LIN {X 0,Y 298.512,Z 418.3,A -85,B 0,C 180,E1 -16399.655,E2 -16399.655} C_VEL
LIN {X 0,Y 298.459,Z 418.309,A -85,B 0,C 180,E1 -16403.598,E2 -16403.598} C_VEL
LIN {X 0,Y 298.488,Z 418.301,A -85,B 0,C 180,E1 -16406.575,E2 -16406.575} C_VEL
LIN {X 0,Y 298.422,Z 418.314,A -85,B 0,C 180,E1 -16409.641,E2 -16409.641} C_VEL
LIN {X 0,Y 298.397,Z 418.313,A -85,B 0,C 180,E1 -16412.8,E2 -16412.8} C_VEL
LIN {X 0,Y 298.466,Z 418.305,A -85,B 0,C 180,E1 -16416.813,E2 -16416.813} C_VEL
LIN {X 0,Y 298.389,Z 418.316,A -85,B 0,C 180,E1 -16421.088,E2 -16421.088} C_VEL
LIN {X 0,Y 298.39,Z 418.318,A -85,B 0,C 180,E1 -16425.042,E2 -16425.042} C_VEL
LIN {X 0,Y 298.389,Z 418.318,A -85,B 0,C 180,E1 -16428.912,E2 -16428.912} C_VEL
LIN {X 0,Y 298.346,Z 418.518,A -85,B 0,C 180,E1 -16432.232,E2 -16432.232} C_VEL
LIN {X 0,Y 298.431,Z 421.494,A -85,B 0,C 180,E1 -16435.584,E2 -16435.584} C_VEL
LIN {X 0,Y 298.189,Z 424.493,A -85,B 0,C 180,E1 -16438.767,E2 -16438.767} C_VEL
LIN {X 0,Y 297.917,Z 427.501,A -85,B 0,C 180,E1 -16441.848,E2 -16441.848} C_VEL
LIN {X 0,Y 297.628,Z 431.178,A -85,B 0,C 180,E1 -16445.445,E2 -16445.445} C_VEL
LIN {X 0,Y 302.039,Z 446.255,A -85,B 0,C 180,E1 -16446.588,E2 -16446.588} C_VEL
LIN {X 0,Y 304.749,Z 458.03,A -85,B 0,C 180,E1 -16447.66,E2 -16447.66} C_VEL
LIN {X 0,Y 306.511,Z 468.932,A -85,B 0,C 180,E1 -16448.83,E2 -16448.83} C_VEL
LIN {X 0,Y 306.054,Z 475.088,A -85,B 0,C 180,E1 -16449.501,E2 -16449.501} C_VEL
LIN {X 0,Y 304.604,Z 485.483,A -85,B 0,C 180,E1 -16450.805,E2 -16450.805} C_VEL
LIN {X 0,Y 303.128,Z 495.965,A -85,B 0,C 180,E1 -16452.458,E2 -16452.458} C_VEL
LIN {X 0,Y 301.615,Z 504.454,A -85,B 0,C 180,E1 -16454.11,E2 -16454.11} C_VEL
LIN {X 0,Y 300.15,Z 512.702,A -85,B 0,C 180,E1 -16456.113,E2 -16456.113} C_VEL
LIN {X 0,Y 299.112,Z 518.344,A -85,B 0,C 180,E1 -16457.792,E2 -16457.792} C_VEL
LIN {X 0,Y 298.123,Z 523.842,A -85,B 0,C 180,E1 -16459.816,E2 -16459.816} C_VEL
LIN {X 0,Y 297.45,Z 528.155,A -85,B 0,C 180,E1 -16461.85,E2 -16461.85} C_VEL
LIN {X 0,Y 297.118,Z 530.806,A -85,B 0,C 180,E1 -16463.447,E2 -16463.447} C_VEL
LIN {X 0,Y 296.785,Z 533.683,A -85,B 0,C 180,E1 -16465.926,E2 -16465.926} C_VEL
LIN {X 0,Y 296.536,Z 535.288,A -85,B 0,C 180,E1 -16468.642,E2 -16468.642} C_VEL
LIN {X 0,Y 296.526,Z 535.518,A -85,B 0,C 180,E1 -16470,E2 -16470} C_VEL
LIN {X 0,Y 296.535,Z 535.326,A -85,B 0,C 180,E1 -16471.358,E2 -16471.358} C_VEL
LIN {X 0,Y 296.78,Z 533.772,A -85,B 0,C 180,E1 -16474.074,E2 -16474.074} C_VEL
LIN {X 0,Y 297.085,Z 531.047,A -85,B 0,C 180,E1 -16476.497,E2 -16476.497} C_VEL
LIN {X 0,Y 297.636,Z 527.076,A -85,B 0,C 180,E1 -16478.829,E2 -16478.829} C_VEL
LIN {X 0,Y 298.406,Z 522.443,A -85,B 0,C 180,E1 -16480.86,E2 -16480.86} C_VEL
LIN {X 0,Y 299.641,Z 515.457,A -85,B 0,C 180,E1 -16483.22,E2 -16483.22} C_VEL
LIN {X 0,Y 301,Z 507.884,A -85,B 0,C 180,E1 -16485.229,E2 -16485.229} C_VEL
LIN {X 0,Y 302.714,Z 498.347,A -85,B 0,C 180,E1 -16487.218,E2 -16487.218} C_VEL
LIN {X 0,Y 304.138,Z 488.507,A -85,B 0,C 180,E1 -16488.876,E2 -16488.876} C_VEL
LIN {X 0,Y 305.739,Z 477.425,A -85,B 0,C 180,E1 -16490.346,E2 -16490.346} C_VEL
LIN {X 0,Y 306.611,Z 469.946,A -85,B 0,C 180,E1 -16491.163,E2 -16491.163} C_VEL
LIN {X 0,Y 304.932,Z 458.822,A -85,B 0,C 180,E1 -16492.374,E2 -16492.374} C_VEL
LIN {X 0,Y 302.205,Z 446.768,A -85,B 0,C 180,E1 -16493.484,E2 -16493.484} C_VEL
LIN {X 0,Y 298.409,Z 433.993,A -85,B 0,C 180,E1 -16494.464,E2 -16494.464} C_VEL
LIN {X 0,Y 297.651,Z 431.164,A -85,B 0,C 180,E1 -16494.685,E2 -16494.685} C_VEL
LIN {X 0,Y 297.91,Z 427.623,A -85,B 0,C 180,E1 -16498.153,E2 -16498.153} C_VEL
LIN {X 0,Y 298.255,Z 423.912,A -85,B 0,C 180,E1 -16501.973,E2 -16501.973} C_VEL
LIN {X 0,Y 298.453,Z 421.544,A -85,B 0,C 180,E1 -16504.494,E2 -16504.494} C_VEL
LIN {X 0,Y 298.4,Z 418.632,A -85,B 0,C 180,E1 -16507.761,E2 -16507.761} C_VEL
LIN {X 0,Y 298.395,Z 418.314,A -85,B 0,C 180,E1 -16509.489,E2 -16509.489} C_VEL
LIN {X 0,Y 298.401,Z 418.314,A -85,B 0,C 180,E1 -16513.103,E2 -16513.103} C_VEL
LIN {X 0,Y 298.405,Z 418.316,A -85,B 0,C 180,E1 -16516.921,E2 -16516.921} C_VEL
LIN {X 0,Y 298.417,Z 418.312,A -85,B 0,C 180,E1 -16521.003,E2 -16521.003} C_VEL
LIN {X 0,Y 298.435,Z 418.309,A -85,B 0,C 180,E1 -16523.932,E2 -16523.932} C_VEL
LIN {X 0,Y 298.398,Z 418.314,A -85,B 0,C 180,E1 -16527.983,E2 -16527.983} C_VEL
LIN {X 0,Y 298.465,Z 418.306,A -85,B 0,C 180,E1 -16531.904,E2 -16531.904} C_VEL
LIN {X 0,Y 298.488,Z 418.302,A -85,B 0,C 180,E1 -16534.924,E2 -16534.924} C_VEL
LIN {X 0,Y 298.46,Z 418.305,A -85,B 0,C 180,E1 -16539.316,E2 -16539.316} C_VEL
LIN {X 0,Y 298.54,Z 418.299,A -85,B 0,C 180,E1 -16542.179,E2 -16542.179} C_VEL
LIN {X 0,Y 298.567,Z 418.29,A -85,B 0,C 180,E1 -16545.385,E2 -16545.385} C_VEL
LIN {X 0,Y 298.597,Z 418.288,A -85,B 0,C 180,E1 -16549.147,E2 -16549.147} C_VEL
LIN {X 0,Y 298.759,Z 418.267,A -85,B 0,C 180,E1 -16551.251,E2 -16551.251} C_VEL
LIN {X 0,Y 298.045,Z 418.361,A -85,B 0,C 180,E1 -16552.375,E2 -16552.375} C_VEL
LIN {X 0,Y 295.086,Z 418.728,A -85,B 0,C 180,E1 -16554.203,E2 -16554.203} C_VEL
LIN {X 0,Y 292.685,Z 419.028,A -85,B 0,C 180,E1 -16555.687,E2 -16555.687} C_VEL
LIN {X 0,Y 291.79,Z 419.135,A -85,B 0,C 180,E1 -16556.838,E2 -16556.838} C_VEL
LIN {X 0,Y 291.788,Z 419.136,A -85,B 0,C 180,E1 -16557.227,E2 -16557.227} C_VEL
LIN {X 0,Y 291.968,Z 419.118,A -85,B 0,C 180,E1 -16560,E2 -16560} C_VEL
LIN {X 0,Y 291.791,Z 419.135,A -85,B 0,C 180,E1 -16562.761,E2 -16562.761} C_VEL
LIN {X 0,Y 291.749,Z 419.142,A -85,B 0,C 180,E1 -16566.918,E2 -16566.918} C_VEL
LIN {X 0,Y 291.632,Z 419.159,A -85,B 0,C 180,E1 -16569.712,E2 -16569.712} C_VEL
LIN {X 0,Y 291.526,Z 419.171,A -85,B 0,C 180,E1 -16573.95,E2 -16573.95} C_VEL
LIN {X 0,Y 291.49,Z 419.174,A -85,B 0,C 180,E1 -16576.818,E2 -16576.818} C_VEL
LIN {X 0,Y 291.453,Z 419.179,A -85,B 0,C 180,E1 -16579.875,E2 -16579.875} C_VEL
LIN {X 0,Y 291.402,Z 419.184,A -85,B 0,C 180,E1 -16584.205,E2 -16584.205} C_VEL
LIN {X 0,Y 291.421,Z 419.186,A -85,B 0,C 180,E1 -16587.272,E2 -16587.272} C_VEL
LIN {X 0,Y 291.336,Z 419.193,A -85,B 0,C 180,E1 -16590.437,E2 -16590.437} C_VEL
LIN {X 0,Y 291.347,Z 419.191,A -85,B 0,C 180,E1 -16593.698,E2 -16593.698} C_VEL
LIN {X 0,Y 291.379,Z 419.191,A -85,B 0,C 180,E1 -16597.254,E2 -16597.254} C_VEL
LIN {X 0,Y 291.335,Z 419.2,A -85,B 0,C 180,E1 -16600.642,E2 -16600.642} C_VEL
LIN {X 0,Y 291.402,Z 419.214,A -85,B 0,C 180,E1 -16603.08,E2 -16603.08} C_VEL
LIN {X 0,Y 291.905,Z 422.504,A -85,B 0,C 180,E1 -16606.244,E2 -16606.244} C_VEL
LIN {X 0,Y 292.649,Z 426.936,A -85,B 0,C 180,E1 -16610.218,E2 -16610.218} C_VEL
LIN {X 0,Y 293,Z 430.406,A -85,B 0,C 180,E1 -16613.154,E2 -16613.154} C_VEL
LIN {X 0,Y 292.811,Z 433.555,A -85,B 0,C 180,E1 -16615.664,E2 -16615.664} C_VEL
LIN {X 0,Y 291.901,Z 439.373,A -85,B 0,C 180,E1 -16620.084,E2 -16620.084} C_VEL
LIN {X 0,Y 291.299,Z 443.573,A -85,B 0,C 180,E1 -16623.212,E2 -16623.212} C_VEL
LIN {X 0,Y 291.037,Z 445.704,A -85,B 0,C 180,E1 -16624.777,E2 -16624.777} C_VEL
LIN {X 0,Y 294.355,Z 459.225,A -85,B 0,C 180,E1 -16625.698,E2 -16625.698} C_VEL
LIN {X 0,Y 296.525,Z 470.949,A -85,B 0,C 180,E1 -16626.687,E2 -16626.687} C_VEL
LIN {X 0,Y 297.887,Z 482.255,A -85,B 0,C 180,E1 -16627.822,E2 -16627.822} C_VEL
LIN {X 0,Y 298.494,Z 491.884,A -85,B 0,C 180,E1 -16628.957,E2 -16628.957} C_VEL
LIN {X 0,Y 296.757,Z 503.417,A -85,B 0,C 180,E1 -16630.457,E2 -16630.457} C_VEL
LIN {X 0,Y 295.242,Z 512.708,A -85,B 0,C 180,E1 -16631.973,E2 -16631.973} C_VEL
LIN {X 0,Y 293.838,Z 521.184,A -85,B 0,C 180,E1 -16633.678,E2 -16633.678} C_VEL
LIN {X 0,Y 292.333,Z 529.457,A -85,B 0,C 180,E1 -16635.734,E2 -16635.734} C_VEL
LIN {X 0,Y 291.102,Z 536.125,A -85,B 0,C 180,E1 -16637.804,E2 -16637.804} C_VEL
LIN {X 0,Y 290.23,Z 542.233,A -85,B 0,C 180,E1 -16640.241,E2 -16640.241} C_VEL
LIN {X 0,Y 289.729,Z 546.204,A -85,B 0,C 180,E1 -16642.333,E2 -16642.333} C_VEL
LIN {X 0,Y 289.479,Z 549.227,A -85,B 0,C 180,E1 -16644.506,E2 -16644.506} C_VEL
LIN {X 0,Y 289.439,Z 551.537,A -85,B 0,C 180,E1 -16647.216,E2 -16647.216} C_VEL
LIN {X 0,Y 289.415,Z 552.145,A -85,B 0,C 180,E1 -16648.608,E2 -16648.608} C_VEL
LIN {X 0,Y 289.437,Z 552.359,A -85,B 0,C 180,E1 -16650,E2 -16650} C_VEL
LIN {X 0,Y 289.415,Z 552.138,A -85,B 0,C 180,E1 -16651.391,E2 -16651.391} C_VEL
LIN {X 0,Y 289.439,Z 551.526,A -85,B 0,C 180,E1 -16652.783,E2 -16652.783} C_VEL
LIN {X 0,Y 289.458,Z 549.252,A -85,B 0,C 180,E1 -16655.451,E2 -16655.451} C_VEL
LIN {X 0,Y 289.728,Z 546.171,A -85,B 0,C 180,E1 -16657.667,E2 -16657.667} C_VEL
LIN {X 0,Y 290.23,Z 542.186,A -85,B 0,C 180,E1 -16659.759,E2 -16659.759} C_VEL
LIN {X 0,Y 291.101,Z 536.059,A -85,B 0,C 180,E1 -16662.195,E2 -16662.195} C_VEL
LIN {X 0,Y 292.333,Z 529.376,A -85,B 0,C 180,E1 -16664.266,E2 -16664.266} C_VEL
LIN {X 0,Y 293.84,Z 521.086,A -85,B 0,C 180,E1 -16666.322,E2 -16666.322} C_VEL
LIN {X 0,Y 295.241,Z 512.583,A -85,B 0,C 180,E1 -16668.026,E2 -16668.026} C_VEL
LIN {X 0,Y 296.742,Z 503.258,A -85,B 0,C 180,E1 -16669.544,E2 -16669.544} C_VEL
LIN {X 0,Y 298.332,Z 493.123,A -85,B 0,C 180,E1 -16670.874,E2 -16670.874} C_VEL
LIN {X 0,Y 298.023,Z 483.792,A -85,B 0,C 180,E1 -16671.985,E2 -16671.985} C_VEL
LIN {X 0,Y 296.647,Z 472.092,A -85,B 0,C 180,E1 -16673.183,E2 -16673.183} C_VEL
LIN {X 0,Y 294.435,Z 459.785,A -85,B 0,C 180,E1 -16674.232,E2 -16674.232} C_VEL
LIN {X 0,Y 291.115,Z 446.415,A -85,B 0,C 180,E1 -16675.161,E2 -16675.161} C_VEL
LIN {X 0,Y 291.029,Z 445.687,A -85,B 0,C 180,E1 -16675.21,E2 -16675.21} C_VEL
LIN {X 0,Y 291.734,Z 440.822,A -85,B 0,C 180,E1 -16678.804,E2 -16678.804} C_VEL
LIN {X 0,Y 292.478,Z 435.563,A -85,B 0,C 180,E1 -16682.752,E2 -16682.752} C_VEL
LIN {X 0,Y 292.995,Z 432.197,A -85,B 0,C 180,E1 -16685.358,E2 -16685.358} C_VEL
LIN {X 0,Y 292.862,Z 428.244,A -85,B 0,C 180,E1 -16688.604,E2 -16688.604} C_VEL
LIN {X 0,Y 292.266,Z 424.569,A -85,B 0,C 180,E1 -16691.803,E2 -16691.803} C_VEL
LIN {X 0,Y 291.576,Z 420.462,A -85,B 0,C 180,E1 -16695.653,E2 -16695.653} C_VEL
LIN {X 0,Y 291.376,Z 419.19,A -85,B 0,C 180,E1 -16696.928,E2 -16696.928} C_VEL
LIN {X 0,Y 291.354,Z 419.196,A -85,B 0,C 180,E1 -16701.158,E2 -16701.158} C_VEL
LIN {X 0,Y 291.362,Z 419.196,A -85,B 0,C 180,E1 -16704.626,E2 -16704.626} C_VEL
LIN {X 0,Y 291.371,Z 419.19,A -85,B 0,C 180,E1 -16707.951,E2 -16707.951} C_VEL
LIN {X 0,Y 291.378,Z 419.19,A -85,B 0,C 180,E1 -16711.158,E2 -16711.158} C_VEL
LIN {X 0,Y 291.413,Z 419.185,A -85,B 0,C 180,E1 -16714.272,E2 -16714.272} C_VEL
LIN {X 0,Y 291.383,Z 419.188,A -85,B 0,C 180,E1 -16717.3,E2 -16717.3} C_VEL
LIN {X 0,Y 291.459,Z 419.18,A -85,B 0,C 180,E1 -16720.27,E2 -16720.27} C_VEL
LIN {X 0,Y 291.556,Z 419.17,A -85,B 0,C 180,E1 -16724.624,E2 -16724.624} C_VEL
LIN {X 0,Y 291.54,Z 419.169,A -85,B 0,C 180,E1 -16728.881,E2 -16728.881} C_VEL
LIN {X 0,Y 291.71,Z 419.147,A -85,B 0,C 180,E1 -16731.689,E2 -16731.689} C_VEL
LIN {X 0,Y 291.632,Z 419.158,A -85,B 0,C 180,E1 -16734.468,E2 -16734.468} C_VEL
LIN {X 0,Y 291.891,Z 419.126,A -85,B 0,C 180,E1 -16738.62,E2 -16738.62} C_VEL
LIN {X 0,Y 291.891,Z 419.124,A -85,B 0,C 180,E1 -16741.38,E2 -16741.38} C_VEL
LIN {X 0,Y 291.748,Z 419.141,A -85,B 0,C 180,E1 -16746.918,E2 -16746.918} C_VEL
LIN {X 0,Y 291.631,Z 419.158,A -85,B 0,C 180,E1 -16749.712,E2 -16749.712} C_VEL
LIN {X 0,Y 291.525,Z 419.173,A -85,B 0,C 180,E1 -16753.95,E2 -16753.95} C_VEL
LIN {X 0,Y 291.488,Z 419.174,A -85,B 0,C 180,E1 -16756.818,E2 -16756.818} C_VEL
LIN {X 0,Y 291.452,Z 419.18,A -85,B 0,C 180,E1 -16759.875,E2 -16759.875} C_VEL
LIN {X 0,Y 291.402,Z 419.186,A -85,B 0,C 180,E1 -16764.205,E2 -16764.205} C_VEL
LIN {X 0,Y 291.422,Z 419.183,A -85,B 0,C 180,E1 -16767.272,E2 -16767.272} C_VEL
LIN {X 0,Y 291.339,Z 419.192,A -85,B 0,C 180,E1 -16770.437,E2 -16770.437} C_VEL
LIN {X 0,Y 291.346,Z 419.195,A -85,B 0,C 180,E1 -16773.698,E2 -16773.698} C_VEL
LIN {X 0,Y 291.396,Z 419.188,A -85,B 0,C 180,E1 -16777.259,E2 -16777.259} C_VEL
LIN {X 0,Y 291.336,Z 419.193,A -85,B 0,C 180,E1 -16780.642,E2 -16780.642} C_VEL
LIN {X 0,Y 291.315,Z 419.197,A -85,B 0,C 180,E1 -16784.397,E2 -16784.397} C_VEL
LIN {X 0,Y 291.328,Z 419.196,A -85,B 0,C 180,E1 -16788.404,E2 -16788.404} C_VEL
LIN {X 0,Y 291.333,Z 419.198,A -85,B 0,C 180,E1 -16791.155,E2 -16791.155} C_VEL
LIN {X 0,Y 291.384,Z 420.19,A -85,B 0,C 180,E1 -16792.916,E2 -16792.916} C_VEL
LIN {X 0,Y 291.348,Z 423.185,A -85,B 0,C 180,E1 -16796.302,E2 -16796.302} C_VEL
LIN {X 0,Y 291.076,Z 426.197,A -85,B 0,C 180,E1 -16799.533,E2 -16799.533} C_VEL
LIN {X 0,Y 290.783,Z 429.984,A -85,B 0,C 180,E1 -16803.414,E2 -16803.414} C_VEL
LIN {X 0,Y 290.64,Z 431.426,A -85,B 0,C 180,E1 -16804.844,E2 -16804.844} C_VEL
LIN {X 0,Y 294.476,Z 444.129,A -85,B 0,C 180,E1 -16805.803,E2 -16805.803} C_VEL
LIN {X 0,Y 297.706,Z 457.33,A -85,B 0,C 180,E1 -16807.026,E2 -16807.026} C_VEL
LIN {X 0,Y 299.647,Z 469.149,A -85,B 0,C 180,E1 -16808.321,E2 -16808.321} C_VEL
LIN {X 0,Y 299.789,Z 472.293,A -85,B 0,C 180,E1 -16808.693,E2 -16808.693} C_VEL
LIN {X 0,Y 298.214,Z 483.339,A -85,B 0,C 180,E1 -16810.018,E2 -16810.018} C_VEL
LIN {X 0,Y 297,Z 492.352,A -85,B 0,C 180,E1 -16811.384,E2 -16811.384} C_VEL
LIN {X 0,Y 295.405,Z 501.444,A -85,B 0,C 180,E1 -16813.056,E2 -16813.056} C_VEL
LIN {X 0,Y 293.703,Z 510.354,A -85,B 0,C 180,E1 -16815.094,E2 -16815.094} C_VEL
LIN {X 0,Y 292.368,Z 517.522,A -85,B 0,C 180,E1 -16817.153,E2 -16817.153} C_VEL
LIN {X 0,Y 291.463,Z 522.355,A -85,B 0,C 180,E1 -16818.878,E2 -16818.878} C_VEL
LIN {X 0,Y 290.623,Z 527.05,A -85,B 0,C 180,E1 -16820.957,E2 -16820.957} C_VEL
LIN {X 0,Y 290.035,Z 531.259,A -85,B 0,C 180,E1 -16823.463,E2 -16823.463} C_VEL
LIN {X 0,Y 289.706,Z 533.888,A -85,B 0,C 180,E1 -16825.827,E2 -16825.827} C_VEL
LIN {X 0,Y 289.457,Z 535.492,A -85,B 0,C 180,E1 -16828.609,E2 -16828.609} C_VEL
LIN {X 0,Y 289.444,Z 535.722,A -85,B 0,C 180,E1 -16830,E2 -16830} C_VEL
LIN {X 0,Y 289.457,Z 535.53,A -85,B 0,C 180,E1 -16831.391,E2 -16831.391} C_VEL
LIN {X 0,Y 289.558,Z 534.943,A -85,B 0,C 180,E1 -16832.783,E2 -16832.783} C_VEL
LIN {X 0,Y 289.701,Z 533.975,A -85,B 0,C 180,E1 -16834.174,E2 -16834.174} C_VEL
LIN {X 0,Y 290.01,Z 531.455,A -85,B 0,C 180,E1 -16836.494,E2 -16836.494} C_VEL
LIN {X 0,Y 290.621,Z 527.279,A -85,B 0,C 180,E1 -16839.044,E2 -16839.044} C_VEL
LIN {X 0,Y 291.438,Z 522.646,A -85,B 0,C 180,E1 -16841.123,E2 -16841.123} C_VEL
LIN {X 0,Y 292.7,Z 515.661,A -85,B 0,C 180,E1 -16843.539,E2 -16843.539} C_VEL
LIN {X 0,Y 294.166,Z 508.085,A -85,B 0,C 180,E1 -16845.592,E2 -16845.592} C_VEL
LIN {X 0,Y 295.941,Z 498.548,A -85,B 0,C 180,E1 -16847.625,E2 -16847.625} C_VEL
LIN {X 0,Y 297.437,Z 488.707,A -85,B 0,C 180,E1 -16849.318,E2 -16849.318} C_VEL
LIN {X 0,Y 299.088,Z 477.624,A -85,B 0,C 180,E1 -16850.819,E2 -16850.819} C_VEL
LIN {X 0,Y 299.869,Z 471.72,A -85,B 0,C 180,E1 -16851.482,E2 -16851.482} C_VEL
LIN {X 0,Y 298.272,Z 460.146,A -85,B 0,C 180,E1 -16852.798,E2 -16852.798} C_VEL
LIN {X 0,Y 295.511,Z 447.816,A -85,B 0,C 180,E1 -16853.997,E2 -16853.997} C_VEL
LIN {X 0,Y 291.757,Z 435.282,A -85,B 0,C 180,E1 -16855.013,E2 -16855.013} C_VEL
LIN {X 0,Y 290.636,Z 431.427,A -85,B 0,C 180,E1 -16855.277,E2 -16855.277} C_VEL
LIN {X 0,Y 290.946,Z 427.824,A -85,B 0,C 180,E1 -16858.889,E2 -16858.889} C_VEL
LIN {X 0,Y 291.256,Z 424.534,A -85,B 0,C 180,E1 -16862.376,E2 -16862.376} C_VEL
LIN {X 0,Y 291.414,Z 421.811,A -85,B 0,C 180,E1 -16865.367,E2 -16865.367} C_VEL
LIN {X 0,Y 291.408,Z 420.148,A -85,B 0,C 180,E1 -16867.262,E2 -16867.262} C_VEL
LIN {X 0,Y 291.33,Z 419.196,A -85,B 0,C 180,E1 -16868.846,E2 -16868.846} C_VEL
LIN {X 0,Y 291.322,Z 419.196,A -85,B 0,C 180,E1 -16872.492,E2 -16872.492} C_VEL
LIN {X 0,Y 291.321,Z 419.196,A -85,B 0,C 180,E1 -16876.364,E2 -16876.364} C_VEL
LIN {X 0,Y 291.39,Z 419.19,A -85,B 0,C 180,E1 -16880.517,E2 -16880.517} C_VEL
LIN {X 0,Y 291.428,Z 419.184,A -85,B 0,C 180,E1 -16882.922,E2 -16882.922} C_VEL
LIN {X 0,Y 291.347,Z 419.195,A -85,B 0,C 180,E1 -16886.302,E2 -16886.302} C_VEL
LIN {X 0,Y 291.389,Z 419.189,A -85,B 0,C 180,E1 -16890.26,E2 -16890.26} C_VEL
LIN {X 0,Y 291.417,Z 419.184,A -85,B 0,C 180,E1 -16894.272,E2 -16894.272} C_VEL
LIN {X 0,Y 291.391,Z 419.185,A -85,B 0,C 180,E1 -16897.3,E2 -16897.3} C_VEL
LIN {X 0,Y 291.461,Z 419.181,A -85,B 0,C 180,E1 -16900.27,E2 -16900.27} C_VEL
LIN {X 0,Y 291.558,Z 419.166,A -85,B 0,C 180,E1 -16904.624,E2 -16904.624} C_VEL
LIN {X 0,Y 291.54,Z 419.167,A -85,B 0,C 180,E1 -16908.881,E2 -16908.881} C_VEL
LIN {X 0,Y 291.712,Z 419.147,A -85,B 0,C 180,E1 -16911.688,E2 -16911.688} C_VEL
LIN {X 0,Y 291.633,Z 419.157,A -85,B 0,C 180,E1 -16914.468,E2 -16914.468} C_VEL
LIN {X 0,Y 291.788,Z 419.136,A -85,B 0,C 180,E1 -16917.227,E2 -16917.227} C_VEL
LIN {X 0,Y 291.322,Z 419.198,A -85,B 0,C 180,E1 -16918.38,E2 -16918.38} C_VEL
LIN {X 0,Y 289.826,Z 419.385,A -85,B 0,C 180,E1 -16919.512,E2 -16919.512} C_VEL
LIN {X 0,Y 285.996,Z 419.862,A -85,B 0,C 180,E1 -16921.782,E2 -16921.782} C_VEL
LIN {X 0,Y 284.788,Z 420.008,A -85,B 0,C 180,E1 -16922.963,E2 -16922.963} C_VEL
LIN {X 0,Y 284.636,Z 420.025,A -85,B 0,C 180,E1 -16923.365,E2 -16923.365} C_VEL
LIN {X 0,Y 284.701,Z 420.02,A -85,B 0,C 180,E1 -16927.09,E2 -16927.09} C_VEL
LIN {X 0,Y 284.57,Z 420.037,A -85,B 0,C 180,E1 -16929.955,E2 -16929.955} C_VEL
LIN {X 0,Y 284.485,Z 420.047,A -85,B 0,C 180,E1 -16934.303,E2 -16934.303} C_VEL
LIN {X 0,Y 284.428,Z 420.056,A -85,B 0,C 180,E1 -16937.248,E2 -16937.248} C_VEL
LIN {X 0,Y 284.381,Z 420.059,A -85,B 0,C 180,E1 -16940.242,E2 -16940.242} C_VEL
LIN {X 0,Y 284.371,Z 420.061,A -85,B 0,C 180,E1 -16943.875,E2 -16943.875} C_VEL
LIN {X 0,Y 284.396,Z 420.061,A -85,B 0,C 180,E1 -16947.172,E2 -16947.172} C_VEL
LIN {X 0,Y 284.296,Z 420.069,A -85,B 0,C 180,E1 -16951.274,E2 -16951.274} C_VEL
LIN {X 0,Y 284.343,Z 420.066,A -85,B 0,C 180,E1 -16955.348,E2 -16955.348} C_VEL
LIN {X 0,Y 284.314,Z 420.068,A -85,B 0,C 180,E1 -16958.169,E2 -16958.169} C_VEL
LIN {X 0,Y 284.334,Z 420.082,A -85,B 0,C 180,E1 -16962.586,E2 -16962.586} C_VEL
LIN {X 0,Y 284.944,Z 423.867,A -85,B 0,C 180,E1 -16966.322,E2 -16966.322} C_VEL
LIN {X 0,Y 285.669,Z 428.1,A -85,B 0,C 180,E1 -16970.234,E2 -16970.234} C_VEL
LIN {X 0,Y 285.981,Z 431.266,A -85,B 0,C 180,E1 -16972.98,E2 -16972.98} C_VEL
LIN {X 0,Y 285.797,Z 434.403,A -85,B 0,C 180,E1 -16975.556,E2 -16975.556} C_VEL
LIN {X 0,Y 284.913,Z 439.712,A -85,B 0,C 180,E1 -16979.695,E2 -16979.695} C_VEL
LIN {X 0,Y 284.161,Z 444.764,A -85,B 0,C 180,E1 -16983.565,E2 -16983.565} C_VEL
LIN {X 0,Y 284.075,Z 445.488,A -85,B 0,C 180,E1 -16984.114,E2 -16984.114} C_VEL
LIN {X 0,Y 287.266,Z 458.185,A -85,B 0,C 180,E1 -16985.007,E2 -16985.007} C_VEL
LIN {X 0,Y 289.635,Z 470.588,A -85,B 0,C 180,E1 -16986.086,E2 -16986.086} C_VEL
LIN {X 0,Y 291.063,Z 482.048,A -85,B 0,C 180,E1 -16987.273,E2 -16987.273} C_VEL
LIN {X 0,Y 291.69,Z 493.113,A -85,B 0,C 180,E1 -16988.628,E2 -16988.628} C_VEL
LIN {X 0,Y 289.859,Z 504.345,A -85,B 0,C 180,E1 -16990.157,E2 -16990.157} C_VEL
LIN {X 0,Y 288.164,Z 514.307,A -85,B 0,C 180,E1 -16991.884,E2 -16991.884} C_VEL
LIN {X 0,Y 286.702,Z 522.472,A -85,B 0,C 180,E1 -16993.626,E2 -16993.626} C_VEL
LIN {X 0,Y 285.188,Z 530.49,A -85,B 0,C 180,E1 -16995.733,E2 -16995.733} C_VEL
LIN {X 0,Y 283.993,Z 536.919,A -85,B 0,C 180,E1 -16997.857,E2 -16997.857} C_VEL
LIN {X 0,Y 283.2,Z 542.029,A -85,B 0,C 180,E1 -16999.996,E2 -16999.996} C_VEL
LIN {X 0,Y 282.685,Z 546.001,A -85,B 0,C 180,E1 -17002.141,E2 -17002.141} C_VEL
LIN {X 0,Y 282.37,Z 549.27,A -85,B 0,C 180,E1 -17004.608,E2 -17004.608} C_VEL
LIN {X 0,Y 282.346,Z 551.333,A -85,B 0,C 180,E1 -17007.146,E2 -17007.146} C_VEL
LIN {X 0,Y 282.338,Z 551.942,A -85,B 0,C 180,E1 -17008.573,E2 -17008.573} C_VEL
LIN {X 0,Y 282.357,Z 552.156,A -85,B 0,C 180,E1 -17010,E2 -17010} C_VEL
LIN {X 0,Y 282.338,Z 551.935,A -85,B 0,C 180,E1 -17011.426,E2 -17011.426} C_VEL
LIN {X 0,Y 282.346,Z 551.322,A -85,B 0,C 180,E1 -17012.853,E2 -17012.853} C_VEL
LIN {X 0,Y 282.35,Z 549.293,A -85,B 0,C 180,E1 -17015.349,E2 -17015.349} C_VEL
LIN {X 0,Y 282.685,Z 545.966,A -85,B 0,C 180,E1 -17017.859,E2 -17017.859} C_VEL
LIN {X 0,Y 283.2,Z 541.979,A -85,B 0,C 180,E1 -17020.004,E2 -17020.004} C_VEL
LIN {X 0,Y 284.129,Z 535.853,A -85,B 0,C 180,E1 -17022.5,E2 -17022.5} C_VEL
LIN {X 0,Y 285.44,Z 529.17,A -85,B 0,C 180,E1 -17024.618,E2 -17024.618} C_VEL
LIN {X 0,Y 287.017,Z 520.879,A -85,B 0,C 180,E1 -17026.721,E2 -17026.721} C_VEL
LIN {X 0,Y 288.474,Z 512.376,A -85,B 0,C 180,E1 -17028.464,E2 -17028.464} C_VEL
LIN {X 0,Y 290.051,Z 503.05,A -85,B 0,C 180,E1 -17030.014,E2 -17030.014} C_VEL
LIN {X 0,Y 291.649,Z 492.913,A -85,B 0,C 180,E1 -17031.375,E2 -17031.375} C_VEL
LIN {X 0,Y 290.98,Z 481.79,A -85,B 0,C 180,E1 -17032.733,E2 -17032.733} C_VEL
LIN {X 0,Y 289.446,Z 469.456,A -85,B 0,C 180,E1 -17033.996,E2 -17033.996} C_VEL
LIN {X 0,Y 286.898,Z 456.681,A -85,B 0,C 180,E1 -17035.078,E2 -17035.078} C_VEL
LIN {X 0,Y 284.075,Z 445.463,A -85,B 0,C 180,E1 -17035.876,E2 -17035.876} C_VEL
LIN {X 0,Y 284.803,Z 440.618,A -85,B 0,C 180,E1 -17039.573,E2 -17039.573} C_VEL
LIN {X 0,Y 285.553,Z 435.93,A -85,B 0,C 180,E1 -17043.196,E2 -17043.196} C_VEL
LIN {X 0,Y 285.951,Z 432.253,A -85,B 0,C 180,E1 -17046.147,E2 -17046.147} C_VEL
LIN {X 0,Y 285.882,Z 429.93,A -85,B 0,C 180,E1 -17048.124,E2 -17048.124} C_VEL
LIN {X 0,Y 285.607,Z 427.452,A -85,B 0,C 180,E1 -17050.286,E2 -17050.286} C_VEL
LIN {X 0,Y 284.832,Z 423.147,A -85,B 0,C 180,E1 -17054.312,E2 -17054.312} C_VEL
LIN {X 0,Y 284.298,Z 420.073,A -85,B 0,C 180,E1 -17057.551,E2 -17057.551} C_VEL
LIN {X 0,Y 284.313,Z 420.072,A -85,B 0,C 180,E1 -17061.831,E2 -17061.831} C_VEL
LIN {X 0,Y 284.309,Z 420.072,A -85,B 0,C 180,E1 -17065.351,E2 -17065.351} C_VEL
LIN {X 0,Y 284.294,Z 420.075,A -85,B 0,C 180,E1 -17068.726,E2 -17068.726} C_VEL
LIN {X 0,Y 284.395,Z 420.062,A -85,B 0,C 180,E1 -17072.827,E2 -17072.827} C_VEL
LIN {X 0,Y 284.368,Z 420.065,A -85,B 0,C 180,E1 -17076.707,E2 -17076.707} C_VEL
LIN {X 0,Y 284.405,Z 420.057,A -85,B 0,C 180,E1 -17081.262,E2 -17081.262} C_VEL
LIN {X 0,Y 284.493,Z 420.049,A -85,B 0,C 180,E1 -17084.459,E2 -17084.459} C_VEL
LIN {X 0,Y 284.491,Z 420.049,A -85,B 0,C 180,E1 -17088.602,E2 -17088.602} C_VEL
LIN {X 0,Y 284.661,Z 420.024,A -85,B 0,C 180,E1 -17091.481,E2 -17091.481} C_VEL
LIN {X 0,Y 284.603,Z 420.033,A -85,B 0,C 180,E1 -17094.331,E2 -17094.331} C_VEL
LIN {X 0,Y 284.857,Z 420.002,A -85,B 0,C 180,E1 -17098.586,E2 -17098.586} C_VEL
LIN {X 0,Y 284.857,Z 420,A -85,B 0,C 180,E1 -17101.414,E2 -17101.414} C_VEL
LIN {X 0,Y 284.7,Z 420.019,A -85,B 0,C 180,E1 -17107.09,E2 -17107.09} C_VEL
LIN {X 0,Y 284.568,Z 420.04,A -85,B 0,C 180,E1 -17109.955,E2 -17109.955} C_VEL
LIN {X 0,Y 284.484,Z 420.048,A -85,B 0,C 180,E1 -17114.303,E2 -17114.303} C_VEL
LIN {X 0,Y 284.427,Z 420.054,A -85,B 0,C 180,E1 -17117.248,E2 -17117.248} C_VEL
LIN {X 0,Y 284.38,Z 420.06,A -85,B 0,C 180,E1 -17120.242,E2 -17120.242} C_VEL
LIN {X 0,Y 284.371,Z 420.064,A -85,B 0,C 180,E1 -17123.876,E2 -17123.876} C_VEL
LIN {X 0,Y 284.397,Z 420.058,A -85,B 0,C 180,E1 -17127.173,E2 -17127.173} C_VEL
LIN {X 0,Y 284.297,Z 420.071,A -85,B 0,C 180,E1 -17131.274,E2 -17131.274} C_VEL
LIN {X 0,Y 284.363,Z 420.064,A -85,B 0,C 180,E1 -17135.354,E2 -17135.354} C_VEL
LIN {X 0,Y 284.325,Z 420.067,A -85,B 0,C 180,E1 -17138.167,E2 -17138.167} C_VEL
LIN {X 0,Y 284.271,Z 420.074,A -85,B 0,C 180,E1 -17142.125,E2 -17142.125} C_VEL
LIN {X 0,Y 284.27,Z 420.075,A -85,B 0,C 180,E1 -17146.192,E2 -17146.192} C_VEL
LIN {X 0,Y 284.307,Z 420.071,A -85,B 0,C 180,E1 -17150.024,E2 -17150.024} C_VEL
LIN {X 0,Y 284.285,Z 420.385,A -85,B 0,C 180,E1 -17151.827,E2 -17151.827} C_VEL
LIN {X 0,Y 284.356,Z 423.38,A -85,B 0,C 180,E1 -17155.357,E2 -17155.357} C_VEL
LIN {X 0,Y 284.108,Z 426.398,A -85,B 0,C 180,E1 -17158.703,E2 -17158.703} C_VEL
LIN {X 0,Y 283.808,Z 429.451,A -85,B 0,C 180,E1 -17161.933,E2 -17161.933} C_VEL
LIN {X 0,Y 283.671,Z 431.624,A -85,B 0,C 180,E1 -17164.175,E2 -17164.175} C_VEL
LIN {X 0,Y 287.749,Z 445.057,A -85,B 0,C 180,E1 -17165.244,E2 -17165.244} C_VEL
LIN {X 0,Y 290.784,Z 457.397,A -85,B 0,C 180,E1 -17166.434,E2 -17166.434} C_VEL
LIN {X 0,Y 292.622,Z 467.644,A -85,B 0,C 180,E1 -17167.587,E2 -17167.587} C_VEL
LIN {X 0,Y 293.138,Z 472.504,A -85,B 0,C 180,E1 -17168.185,E2 -17168.185} C_VEL
LIN {X 0,Y 291.562,Z 483.547,A -85,B 0,C 180,E1 -17169.542,E2 -17169.542} C_VEL
LIN {X 0,Y 290.196,Z 493.082,A -85,B 0,C 180,E1 -17171.028,E2 -17171.028} C_VEL
LIN {X 0,Y 288.301,Z 503.272,A -85,B 0,C 180,E1 -17172.991,E2 -17172.991} C_VEL
LIN {X 0,Y 286.59,Z 511.889,A -85,B 0,C 180,E1 -17175.079,E2 -17175.079} C_VEL
LIN {X 0,Y 285.237,Z 518.756,A -85,B 0,C 180,E1 -17177.188,E2 -17177.188} C_VEL
LIN {X 0,Y 284.167,Z 524.253,A -85,B 0,C 180,E1 -17179.31,E2 -17179.31} C_VEL
LIN {X 0,Y 283.397,Z 528.565,A -85,B 0,C 180,E1 -17181.443,E2 -17181.443} C_VEL
LIN {X 0,Y 282.923,Z 531.752,A -85,B 0,C 180,E1 -17183.53,E2 -17183.53} C_VEL
LIN {X 0,Y 282.63,Z 534.092,A -85,B 0,C 180,E1 -17185.722,E2 -17185.722} C_VEL
LIN {X 0,Y 282.493,Z 535.084,A -85,B 0,C 180,E1 -17187.148,E2 -17187.148} C_VEL
LIN {X 0,Y 282.364,Z 535.925,A -85,B 0,C 180,E1 -17190,E2 -17190} C_VEL
LIN {X 0,Y 282.38,Z 535.733,A -85,B 0,C 180,E1 -17191.426,E2 -17191.426} C_VEL
LIN {X 0,Y 282.491,Z 535.146,A -85,B 0,C 180,E1 -17192.852,E2 -17192.852} C_VEL
LIN {X 0,Y 282.625,Z 534.178,A -85,B 0,C 180,E1 -17194.278,E2 -17194.278} C_VEL
LIN {X 0,Y 282.942,Z 531.848,A -85,B 0,C 180,E1 -17196.504,E2 -17196.504} C_VEL
LIN {X 0,Y 283.397,Z 528.762,A -85,B 0,C 180,E1 -17198.557,E2 -17198.557} C_VEL
LIN {X 0,Y 284.13,Z 524.51,A -85,B 0,C 180,E1 -17200.691,E2 -17200.691} C_VEL
LIN {X 0,Y 285.386,Z 518.07,A -85,B 0,C 180,E1 -17203.167,E2 -17203.167} C_VEL
LIN {X 0,Y 286.765,Z 510.99,A -85,B 0,C 180,E1 -17205.276,E2 -17205.276} C_VEL
LIN {X 0,Y 288.552,Z 502.165,A -85,B 0,C 180,E1 -17207.359,E2 -17207.359} C_VEL
LIN {X 0,Y 290.088,Z 492.988,A -85,B 0,C 180,E1 -17209.115,E2 -17209.115} C_VEL
LIN {X 0,Y 291.674,Z 483.081,A -85,B 0,C 180,E1 -17210.634,E2 -17210.634} C_VEL
LIN {X 0,Y 293.119,Z 473.494,A -85,B 0,C 180,E1 -17211.817,E2 -17211.817} C_VEL
LIN {X 0,Y 292.163,Z 464.863,A -85,B 0,C 180,E1 -17212.865,E2 -17212.865} C_VEL
LIN {X 0,Y 289.961,Z 453.507,A -85,B 0,C 180,E1 -17214.084,E2 -17214.084} C_VEL
LIN {X 0,Y 286.608,Z 441.206,A -85,B 0,C 180,E1 -17215.21,E2 -17215.21} C_VEL
LIN {X 0,Y 283.661,Z 431.608,A -85,B 0,C 180,E1 -17215.968,E2 -17215.968} C_VEL
LIN {X 0,Y 284.021,Z 427.719,A -85,B 0,C 180,E1 -17219.995,E2 -17219.995} C_VEL
LIN {X 0,Y 284.25,Z 425.011,A -85,B 0,C 180,E1 -17222.953,E2 -17222.953} C_VEL
LIN {X 0,Y 284.38,Z 422.009,A -85,B 0,C 180,E1 -17226.379,E2 -17226.379} C_VEL
LIN {X 0,Y 284.311,Z 420.497,A -85,B 0,C 180,E1 -17228.169,E2 -17228.169} C_VEL
LIN {X 0,Y 284.307,Z 420.069,A -85,B 0,C 180,E1 -17229.995,E2 -17229.995} C_VEL
LIN {X 0,Y 284.268,Z 420.073,A -85,B 0,C 180,E1 -17234.195,E2 -17234.195} C_VEL
LIN {X 0,Y 284.275,Z 420.074,A -85,B 0,C 180,E1 -17238.125,E2 -17238.125} C_VEL
LIN {X 0,Y 284.338,Z 420.066,A -85,B 0,C 180,E1 -17242.274,E2 -17242.274} C_VEL
LIN {X 0,Y 284.326,Z 420.067,A -85,B 0,C 180,E1 -17245.353,E2 -17245.353} C_VEL
LIN {X 0,Y 284.298,Z 420.072,A -85,B 0,C 180,E1 -17248.726,E2 -17248.726} C_VEL
LIN {X 0,Y 284.398,Z 420.058,A -85,B 0,C 180,E1 -17252.827,E2 -17252.827} C_VEL
LIN {X 0,Y 284.371,Z 420.062,A -85,B 0,C 180,E1 -17256.707,E2 -17256.707} C_VEL
LIN {X 0,Y 284.406,Z 420.056,A -85,B 0,C 180,E1 -17261.262,E2 -17261.262} C_VEL
LIN {X 0,Y 284.495,Z 420.046,A -85,B 0,C 180,E1 -17264.459,E2 -17264.459} C_VEL
LIN {X 0,Y 284.491,Z 420.046,A -85,B 0,C 180,E1 -17268.601,E2 -17268.601} C_VEL
LIN {X 0,Y 284.662,Z 420.024,A -85,B 0,C 180,E1 -17271.481,E2 -17271.481} C_VEL
LIN {X 0,Y 284.604,Z 420.033,A -85,B 0,C 180,E1 -17274.331,E2 -17274.331} C_VEL
LIN {X 0,Y 284.857,Z 420,A -85,B 0,C 180,E1 -17278.586,E2 -17278.586} C_VEL
LIN {X 0,Y 284.858,Z 420.002,A -85,B 0,C 180,E1 -17281.414,E2 -17281.414} C_VEL
LIN {X 0,Y 284.636,Z 420.025,A -85,B 0,C 180,E1 -17283.365,E2 -17283.365} C_VEL
LIN {X 0,Y 283.856,Z 420.125,A -85,B 0,C 180,E1 -17284.546,E2 -17284.546} C_VEL
LIN {X 0,Y 281.064,Z 420.473,A -85,B 0,C 180,E1 -17286.475,E2 -17286.475} C_VEL
LIN {X 0,Y 277.932,Z 420.863,A -85,B 0,C 180,E1 -17288.842,E2 -17288.842} C_VEL
LIN {X 0,Y 277.563,Z 420.908,A -85,B 0,C 180,E1 -17289.659,E2 -17289.659} C_VEL
LIN {X 0,Y 277.438,Z 420.924,A -85,B 0,C 180,E1 -17294.674,E2 -17294.674} C_VEL
LIN {X 0,Y 277.347,Z 420.939,A -85,B 0,C 180,E1 -17299.234,E2 -17299.234} C_VEL
LIN {X 0,Y 277.321,Z 420.938,A -85,B 0,C 180,E1 -17304.17,E2 -17304.17} C_VEL
LIN {X 0,Y 277.325,Z 420.94,A -85,B 0,C 180,E1 -17307.504,E2 -17307.504} C_VEL
LIN {X 0,Y 277.274,Z 420.946,A -85,B 0,C 180,E1 -17310.481,E2 -17310.481} C_VEL
LIN {X 0,Y 277.249,Z 420.947,A -85,B 0,C 180,E1 -17313.896,E2 -17313.896} C_VEL
LIN {X 0,Y 277.27,Z 420.947,A -85,B 0,C 180,E1 -17317.469,E2 -17317.469} C_VEL
LIN {X 0,Y 277.258,Z 421.046,A -85,B 0,C 180,E1 -17322.165,E2 -17322.165} C_VEL
LIN {X 0,Y 277.759,Z 423.905,A -85,B 0,C 180,E1 -17325.111,E2 -17325.111} C_VEL
LIN {X 0,Y 278.453,Z 428.153,A -85,B 0,C 180,E1 -17329.217,E2 -17329.217} C_VEL
LIN {X 0,Y 278.968,Z 432.126,A -85,B 0,C 180,E1 -17332.798,E2 -17332.798} C_VEL
LIN {X 0,Y 278.791,Z 435.264,A -85,B 0,C 180,E1 -17335.445,E2 -17335.445} C_VEL
LIN {X 0,Y 277.887,Z 440.454,A -85,B 0,C 180,E1 -17339.614,E2 -17339.614} C_VEL
LIN {X 0,Y 277.134,Z 445.282,A -85,B 0,C 180,E1 -17343.417,E2 -17343.417} C_VEL
LIN {X 0,Y 279.782,Z 455.675,A -85,B 0,C 180,E1 -17344.164,E2 -17344.164} C_VEL
LIN {X 0,Y 282.423,Z 468.047,A -85,B 0,C 180,E1 -17345.243,E2 -17345.243} C_VEL
LIN {X 0,Y 284.058,Z 480.175,A -85,B 0,C 180,E1 -17346.499,E2 -17346.499} C_VEL
LIN {X 0,Y 284.86,Z 491.573,A -85,B 0,C 180,E1 -17347.912,E2 -17347.912} C_VEL
LIN {X 0,Y 284.677,Z 495.642,A -85,B 0,C 180,E1 -17348.455,E2 -17348.455} C_VEL
LIN {X 0,Y 282.75,Z 506.287,A -85,B 0,C 180,E1 -17350.015,E2 -17350.015} C_VEL
LIN {X 0,Y 281.186,Z 515.254,A -85,B 0,C 180,E1 -17351.66,E2 -17351.66} C_VEL
LIN {X 0,Y 279.573,Z 523.758,A -85,B 0,C 180,E1 -17353.572,E2 -17353.572} C_VEL
LIN {X 0,Y 278.04,Z 531.444,A -85,B 0,C 180,E1 -17355.732,E2 -17355.732} C_VEL
LIN {X 0,Y 277.001,Z 536.714,A -85,B 0,C 180,E1 -17357.546,E2 -17357.546} C_VEL
LIN {X 0,Y 276.186,Z 541.825,A -85,B 0,C 180,E1 -17359.739,E2 -17359.739} C_VEL
LIN {X 0,Y 275.617,Z 545.796,A -85,B 0,C 180,E1 -17361.938,E2 -17361.938} C_VEL
LIN {X 0,Y 275.263,Z 549.311,A -85,B 0,C 180,E1 -17364.714,E2 -17364.714} C_VEL
LIN {X 0,Y 275.256,Z 551.13,A -85,B 0,C 180,E1 -17367.073,E2 -17367.073} C_VEL
LIN {X 0,Y 275.263,Z 551.739,A -85,B 0,C 180,E1 -17368.537,E2 -17368.537} C_VEL
LIN {X 0,Y 275.278,Z 551.953,A -85,B 0,C 180,E1 -17370,E2 -17370} C_VEL
LIN {X 0,Y 275.263,Z 551.731,A -85,B 0,C 180,E1 -17371.463,E2 -17371.463} C_VEL
LIN {X 0,Y 275.255,Z 551.118,A -85,B 0,C 180,E1 -17372.927,E2 -17372.927} C_VEL
LIN {X 0,Y 275.253,Z 549.313,A -85,B 0,C 180,E1 -17375.262,E2 -17375.262} C_VEL
LIN {X 0,Y 275.616,Z 545.76,A -85,B 0,C 180,E1 -17378.062,E2 -17378.062} C_VEL
LIN {X 0,Y 276.186,Z 541.774,A -85,B 0,C 180,E1 -17380.261,E2 -17380.261} C_VEL
LIN {X 0,Y 277.171,Z 535.646,A -85,B 0,C 180,E1 -17382.819,E2 -17382.819} C_VEL
LIN {X 0,Y 278.563,Z 528.964,A -85,B 0,C 180,E1 -17384.987,E2 -17384.987} C_VEL
LIN {X 0,Y 280.208,Z 520.672,A -85,B 0,C 180,E1 -17387.14,E2 -17387.14} C_VEL
LIN {X 0,Y 281.697,Z 512.167,A -85,B 0,C 180,E1 -17388.925,E2 -17388.925} C_VEL
LIN {X 0,Y 283.57,Z 501.665,A -85,B 0,C 180,E1 -17390.681,E2 -17390.681} C_VEL
LIN {X 0,Y 284.842,Z 494.131,A -85,B 0,C 180,E1 -17391.722,E2 -17391.722} C_VEL
LIN {X 0,Y 284.33,Z 483.363,A -85,B 0,C 180,E1 -17393.103,E2 -17393.103} C_VEL
LIN {X 0,Y 282.906,Z 471.207,A -85,B 0,C 180,E1 -17394.418,E2 -17394.418} C_VEL
LIN {X 0,Y 280.355,Z 458.105,A -85,B 0,C 180,E1 -17395.613,E2 -17395.613} C_VEL
LIN {X 0,Y 277.127,Z 445.238,A -85,B 0,C 180,E1 -17396.588,E2 -17396.588} C_VEL
LIN {X 0,Y 277.991,Z 439.975,A -85,B 0,C 180,E1 -17400.732,E2 -17400.732} C_VEL
LIN {X 0,Y 278.792,Z 435.197,A -85,B 0,C 180,E1 -17404.555,E2 -17404.555} C_VEL
LIN {X 0,Y 278.915,Z 432.062,A -85,B 0,C 180,E1 -17407.21,E2 -17407.21} C_VEL
LIN {X 0,Y 278.48,Z 428.095,A -85,B 0,C 180,E1 -17410.79,E2 -17410.79} C_VEL
LIN {X 0,Y 277.691,Z 423.592,A -85,B 0,C 180,E1 -17415.125,E2 -17415.125} C_VEL
LIN {X 0,Y 277.236,Z 420.952,A -85,B 0,C 180,E1 -17418.024,E2 -17418.024} C_VEL
LIN {X 0,Y 277.269,Z 420.951,A -85,B 0,C 180,E1 -17422.531,E2 -17422.531} C_VEL
LIN {X 0,Y 277.248,Z 420.951,A -85,B 0,C 180,E1 -17426.104,E2 -17426.104} C_VEL
LIN {X 0,Y 277.262,Z 420.948,A -85,B 0,C 180,E1 -17429.539,E2 -17429.539} C_VEL
LIN {X 0,Y 277.357,Z 420.938,A -85,B 0,C 180,E1 -17432.864,E2 -17432.864} C_VEL
LIN {X 0,Y 277.329,Z 420.939,A -85,B 0,C 180,E1 -17436.08,E2 -17436.08} C_VEL
LIN {X 0,Y 277.346,Z 420.94,A -85,B 0,C 180,E1 -17440.766,E2 -17440.766} C_VEL
LIN {X 0,Y 277.436,Z 420.925,A -85,B 0,C 180,E1 -17445.326,E2 -17445.326} C_VEL
LIN {X 0,Y 277.509,Z 420.916,A -85,B 0,C 180,E1 -17449.789,E2 -17449.789} C_VEL
LIN {X 0,Y 277.655,Z 420.897,A -85,B 0,C 180,E1 -17452.729,E2 -17452.729} C_VEL
LIN {X 0,Y 277.823,Z 420.879,A -85,B 0,C 180,E1 -17458.551,E2 -17458.551} C_VEL
LIN {X 0,Y 277.823,Z 420.876,A -85,B 0,C 180,E1 -17461.45,E2 -17461.45} C_VEL
LIN {X 0,Y 277.655,Z 420.897,A -85,B 0,C 180,E1 -17467.271,E2 -17467.271} C_VEL
LIN {X 0,Y 277.509,Z 420.918,A -85,B 0,C 180,E1 -17470.211,E2 -17470.211} C_VEL
LIN {X 0,Y 277.437,Z 420.925,A -85,B 0,C 180,E1 -17474.674,E2 -17474.674} C_VEL
LIN {X 0,Y 277.346,Z 420.934,A -85,B 0,C 180,E1 -17479.234,E2 -17479.234} C_VEL
LIN {X 0,Y 277.321,Z 420.94,A -85,B 0,C 180,E1 -17484.171,E2 -17484.171} C_VEL
LIN {X 0,Y 277.326,Z 420.941,A -85,B 0,C 180,E1 -17487.505,E2 -17487.505} C_VEL
LIN {X 0,Y 277.273,Z 420.944,A -85,B 0,C 180,E1 -17490.481,E2 -17490.481} C_VEL
LIN {X 0,Y 277.256,Z 420.949,A -85,B 0,C 180,E1 -17493.895,E2 -17493.895} C_VEL
LIN {X 0,Y 277.283,Z 420.947,A -85,B 0,C 180,E1 -17497.467,E2 -17497.467} C_VEL
LIN {X 0,Y 277.211,Z 420.956,A -85,B 0,C 180,E1 -17501.237,E2 -17501.237} C_VEL
LIN {X 0,Y 277.218,Z 420.956,A -85,B 0,C 180,E1 -17505.223,E2 -17505.223} C_VEL
LIN {X 0,Y 277.224,Z 420.954,A -85,B 0,C 180,E1 -17509.512,E2 -17509.512} C_VEL
LIN {X 0,Y 277.227,Z 420.954,A -85,B 0,C 180,E1 -17510.671,E2 -17510.671} C_VEL
LIN {X 0,Y 277.32,Z 422.07,A -85,B 0,C 180,E1 -17512.539,E2 -17512.539} C_VEL
LIN {X 0,Y 277.349,Z 423.567,A -85,B 0,C 180,E1 -17514.351,E2 -17514.351} C_VEL
LIN {X 0,Y 277.147,Z 426.589,A -85,B 0,C 180,E1 -17517.824,E2 -17517.824} C_VEL
LIN {X 0,Y 276.834,Z 429.658,A -85,B 0,C 180,E1 -17521.161,E2 -17521.161} C_VEL
LIN {X 0,Y 276.697,Z 431.833,A -85,B 0,C 180,E1 -17523.459,E2 -17523.459} C_VEL
LIN {X 0,Y 281.142,Z 446.408,A -85,B 0,C 180,E1 -17524.695,E2 -17524.695} C_VEL
LIN {X 0,Y 284.22,Z 458.995,A -85,B 0,C 180,E1 -17525.975,E2 -17525.975} C_VEL
LIN {X 0,Y 286.034,Z 469.583,A -85,B 0,C 180,E1 -17527.233,E2 -17527.233} C_VEL
LIN {X 0,Y 286.395,Z 474.279,A -85,B 0,C 180,E1 -17527.834,E2 -17527.834} C_VEL
LIN {X 0,Y 284.718,Z 484.939,A -85,B 0,C 180,E1 -17529.217,E2 -17529.217} C_VEL
LIN {X 0,Y 283.163,Z 495.208,A -85,B 0,C 180,E1 -17530.91,E2 -17530.91} C_VEL
LIN {X 0,Y 281.537,Z 503.478,A -85,B 0,C 180,E1 -17532.569,E2 -17532.569} C_VEL
LIN {X 0,Y 279.745,Z 512.095,A -85,B 0,C 180,E1 -17534.705,E2 -17534.705} C_VEL
LIN {X 0,Y 278.322,Z 518.962,A -85,B 0,C 180,E1 -17536.864,E2 -17536.864} C_VEL
LIN {X 0,Y 277.18,Z 524.458,A -85,B 0,C 180,E1 -17539.038,E2 -17539.038} C_VEL
LIN {X 0,Y 276.387,Z 528.77,A -85,B 0,C 180,E1 -17541.224,E2 -17541.224} C_VEL
LIN {X 0,Y 275.832,Z 532.199,A -85,B 0,C 180,E1 -17543.564,E2 -17543.564} C_VEL
LIN {X 0,Y 275.557,Z 534.297,A -85,B 0,C 180,E1 -17545.612,E2 -17545.612} C_VEL
LIN {X 0,Y 275.427,Z 535.288,A -85,B 0,C 180,E1 -17547.075,E2 -17547.075} C_VEL
LIN {X 0,Y 275.286,Z 536.129,A -85,B 0,C 180,E1 -17550,E2 -17550} C_VEL
LIN {X 0,Y 275.306,Z 535.936,A -85,B 0,C 180,E1 -17551.463,E2 -17551.463} C_VEL
LIN {X 0,Y 275.425,Z 535.349,A -85,B 0,C 180,E1 -17552.925,E2 -17552.925} C_VEL
LIN {X 0,Y 275.552,Z 534.382,A -85,B 0,C 180,E1 -17554.388,E2 -17554.388} C_VEL
LIN {X 0,Y 275.872,Z 532.245,A -85,B 0,C 180,E1 -17556.51,E2 -17556.51} C_VEL
LIN {X 0,Y 276.386,Z 528.965,A -85,B 0,C 180,E1 -17558.776,E2 -17558.776} C_VEL
LIN {X 0,Y 277.148,Z 524.713,A -85,B 0,C 180,E1 -17560.964,E2 -17560.964} C_VEL
LIN {X 0,Y 278.483,Z 518.272,A -85,B 0,C 180,E1 -17563.5,E2 -17563.5} C_VEL
LIN {X 0,Y 279.917,Z 511.192,A -85,B 0,C 180,E1 -17565.659,E2 -17565.659} C_VEL
LIN {X 0,Y 281.796,Z 502.366,A -85,B 0,C 180,E1 -17567.789,E2 -17567.789} C_VEL
LIN {X 0,Y 283.433,Z 492.836,A -85,B 0,C 180,E1 -17569.649,E2 -17569.649} C_VEL
LIN {X 0,Y 285.231,Z 481.993,A -85,B 0,C 180,E1 -17571.312,E2 -17571.312} C_VEL
LIN {X 0,Y 286.451,Z 473.696,A -85,B 0,C 180,E1 -17572.352,E2 -17572.352} C_VEL
LIN {X 0,Y 284.81,Z 461.921,A -85,B 0,C 180,E1 -17573.808,E2 -17573.808} C_VEL
LIN {X 0,Y 282.226,Z 450.355,A -85,B 0,C 180,E1 -17575.046,E2 -17575.046} C_VEL
LIN {X 0,Y 278.546,Z 437.681,A -85,B 0,C 180,E1 -17576.198,E2 -17576.198} C_VEL
LIN {X 0,Y 276.715,Z 431.839,A -85,B 0,C 180,E1 -17576.659,E2 -17576.659} C_VEL
LIN {X 0,Y 277,Z 428.233,A -85,B 0,C 180,E1 -17580.493,E2 -17580.493} C_VEL
LIN {X 0,Y 277.282,Z 425.224,A -85,B 0,C 180,E1 -17583.891,E2 -17583.891} C_VEL
LIN {X 0,Y 277.341,Z 422.2,A -85,B 0,C 180,E1 -17587.458,E2 -17587.458} C_VEL
LIN {X 0,Y 277.235,Z 420.951,A -85,B 0,C 180,E1 -17589.328,E2 -17589.328} C_VEL
LIN {X 0,Y 277.219,Z 420.952,A -85,B 0,C 180,E1 -17593.197,E2 -17593.197} C_VEL
LIN {X 0,Y 277.22,Z 420.952,A -85,B 0,C 180,E1 -17597.324,E2 -17597.324} C_VEL
LIN {X 0,Y 277.278,Z 420.944,A -85,B 0,C 180,E1 -17601.79,E2 -17601.79} C_VEL
LIN {X 0,Y 277.306,Z 420.943,A -85,B 0,C 180,E1 -17604.344,E2 -17604.344} C_VEL
LIN {X 0,Y 277.247,Z 420.948,A -85,B 0,C 180,E1 -17607.837,E2 -17607.837} C_VEL
LIN {X 0,Y 277.273,Z 420.944,A -85,B 0,C 180,E1 -17611.21,E2 -17611.21} C_VEL
LIN {X 0,Y 277.315,Z 420.94,A -85,B 0,C 180,E1 -17614.48,E2 -17614.48} C_VEL
LIN {X 0,Y 277.293,Z 420.942,A -85,B 0,C 180,E1 -17617.655,E2 -17617.655} C_VEL
LIN {X 0,Y 277.348,Z 420.936,A -85,B 0,C 180,E1 -17620.766,E2 -17620.766} C_VEL
LIN {X 0,Y 277.437,Z 420.923,A -85,B 0,C 180,E1 -17625.326,E2 -17625.326} C_VEL
LIN {X 0,Y 277.509,Z 420.918,A -85,B 0,C 180,E1 -17629.789,E2 -17629.789} C_VEL
LIN {X 0,Y 277.656,Z 420.897,A -85,B 0,C 180,E1 -17632.729,E2 -17632.729} C_VEL
LIN {X 0,Y 277.823,Z 420.876,A -85,B 0,C 180,E1 -17638.55,E2 -17638.55} C_VEL
LIN {X 0,Y 277.824,Z 420.878,A -85,B 0,C 180,E1 -17641.449,E2 -17641.449} C_VEL
LIN {X 0,Y 277.656,Z 420.899,A -85,B 0,C 180,E1 -17647.271,E2 -17647.271} C_VEL
LIN {X 0,Y 277.563,Z 420.908,A -85,B 0,C 180,E1 -17649.659,E2 -17649.659} C_VEL
LIN {X 0,Y 276.804,Z 421.004,A -85,B 0,C 180,E1 -17650.868,E2 -17650.868} C_VEL
LIN {X 0,Y 273.923,Z 421.366,A -85,B 0,C 180,E1 -17652.839,E2 -17652.839} C_VEL
LIN {X 0,Y 271.519,Z 421.666,A -85,B 0,C 180,E1 -17654.44,E2 -17654.44} C_VEL
LIN {X 0,Y 270.47,Z 421.795,A -85,B 0,C 180,E1 -17655.68,E2 -17655.68} C_VEL
LIN {X 0,Y 270.372,Z 421.805,A -85,B 0,C 180,E1 -17656.101,E2 -17656.101} C_VEL
LIN {X 0,Y 270.295,Z 421.814,A -85,B 0,C 180,E1 -17660.602,E2 -17660.602} C_VEL
LIN {X 0,Y 270.276,Z 421.816,A -85,B 0,C 180,E1 -17664.585,E2 -17664.585} C_VEL
LIN {X 0,Y 270.271,Z 421.816,A -85,B 0,C 180,E1 -17667.909,E2 -17667.909} C_VEL
LIN {X 0,Y 270.186,Z 421.826,A -85,B 0,C 180,E1 -17671.348,E2 -17671.348} C_VEL
LIN {X 0,Y 270.204,Z 421.827,A -85,B 0,C 180,E1 -17674.905,E2 -17674.905} C_VEL
LIN {X 0,Y 270.199,Z 421.83,A -85,B 0,C 180,E1 -17678.71,E2 -17678.71} C_VEL
LIN {X 0,Y 270.223,Z 421.998,A -85,B 0,C 180,E1 -17681.717,E2 -17681.717} C_VEL
LIN {X 0,Y 270.825,Z 425.583,A -85,B 0,C 180,E1 -17685.52,E2 -17685.52} C_VEL
LIN {X 0,Y 271.524,Z 429.815,A -85,B 0,C 180,E1 -17689.677,E2 -17689.677} C_VEL
LIN {X 0,Y 271.931,Z 433.702,A -85,B 0,C 180,E1 -17693.244,E2 -17693.244} C_VEL
LIN {X 0,Y 271.619,Z 436.794,A -85,B 0,C 180,E1 -17695.892,E2 -17695.892} C_VEL
LIN {X 0,Y 270.657,Z 442.301,A -85,B 0,C 180,E1 -17700.438,E2 -17700.438} C_VEL
LIN {X 0,Y 270.176,Z 445.061,A -85,B 0,C 180,E1 -17702.673,E2 -17702.673} C_VEL
LIN {X 0,Y 273.654,Z 458.531,A -85,B 0,C 180,E1 -17703.721,E2 -17703.721} C_VEL
LIN {X 0,Y 276.118,Z 471.062,A -85,B 0,C 180,E1 -17704.914,E2 -17704.914} C_VEL
LIN {X 0,Y 277.559,Z 483.196,A -85,B 0,C 180,E1 -17706.274,E2 -17706.274} C_VEL
LIN {X 0,Y 278.118,Z 492.859,A -85,B 0,C 180,E1 -17707.551,E2 -17707.551} C_VEL
LIN {X 0,Y 277.619,Z 498.03,A -85,B 0,C 180,E1 -17708.27,E2 -17708.27} C_VEL
LIN {X 0,Y 275.681,Z 508.197,A -85,B 0,C 180,E1 -17709.869,E2 -17709.869} C_VEL
LIN {X 0,Y 274.04,Z 517,A -85,B 0,C 180,E1 -17711.604,E2 -17711.604} C_VEL
LIN {X 0,Y 272.443,Z 524.931,A -85,B 0,C 180,E1 -17713.515,E2 -17713.515} C_VEL
LIN {X 0,Y 270.916,Z 532.363,A -85,B 0,C 180,E1 -17715.733,E2 -17715.733} C_VEL
LIN {X 0,Y 269.708,Z 538.334,A -85,B 0,C 180,E1 -17717.968,E2 -17717.968} C_VEL
LIN {X 0,Y 268.947,Z 543.056,A -85,B 0,C 180,E1 -17720.22,E2 -17720.22} C_VEL
LIN {X 0,Y 268.421,Z 546.666,A -85,B 0,C 180,E1 -17722.477,E2 -17722.477} C_VEL
LIN {X 0,Y 268.179,Z 549.304,A -85,B 0,C 180,E1 -17724.775,E2 -17724.775} C_VEL
LIN {X 0,Y 268.168,Z 550.926,A -85,B 0,C 180,E1 -17726.995,E2 -17726.995} C_VEL
LIN {X 0,Y 268.189,Z 551.535,A -85,B 0,C 180,E1 -17728.498,E2 -17728.498} C_VEL
LIN {X 0,Y 268.202,Z 551.749,A -85,B 0,C 180,E1 -17730,E2 -17730} C_VEL
LIN {X 0,Y 268.189,Z 551.527,A -85,B 0,C 180,E1 -17731.501,E2 -17731.501} C_VEL
LIN {X 0,Y 268.167,Z 550.913,A -85,B 0,C 180,E1 -17733.004,E2 -17733.004} C_VEL
LIN {X 0,Y 268.169,Z 549.304,A -85,B 0,C 180,E1 -17735.2,E2 -17735.2} C_VEL
LIN {X 0,Y 268.562,Z 545.554,A -85,B 0,C 180,E1 -17738.275,E2 -17738.275} C_VEL
LIN {X 0,Y 269.17,Z 541.568,A -85,B 0,C 180,E1 -17740.531,E2 -17740.531} C_VEL
LIN {X 0,Y 270.228,Z 535.44,A -85,B 0,C 180,E1 -17743.154,E2 -17743.154} C_VEL
LIN {X 0,Y 271.701,Z 528.757,A -85,B 0,C 180,E1 -17745.375,E2 -17745.375} C_VEL
LIN {X 0,Y 273.415,Z 520.466,A -85,B 0,C 180,E1 -17747.579,E2 -17747.579} C_VEL
LIN {X 0,Y 274.958,Z 511.959,A -85,B 0,C 180,E1 -17749.407,E2 -17749.407} C_VEL
LIN {X 0,Y 276.948,Z 501.458,A -85,B 0,C 180,E1 -17751.199,E2 -17751.199} C_VEL
LIN {X 0,Y 278.097,Z 493.917,A -85,B 0,C 180,E1 -17752.276,E2 -17752.276} C_VEL
LIN {X 0,Y 277.515,Z 483.144,A -85,B 0,C 180,E1 -17753.704,E2 -17753.704} C_VEL
LIN {X 0,Y 276.069,Z 470.983,A -85,B 0,C 180,E1 -17755.064,E2 -17755.064} C_VEL
LIN {X 0,Y 273.535,Z 458.023,A -85,B 0,C 180,E1 -17756.29,E2 -17756.29} C_VEL
LIN {X 0,Y 270.201,Z 445.018,A -85,B 0,C 180,E1 -17757.327,E2 -17757.327} C_VEL
LIN {X 0,Y 271.022,Z 440.208,A -85,B 0,C 180,E1 -17761.24,E2 -17761.24} C_VEL
LIN {X 0,Y 271.771,Z 436.034,A -85,B 0,C 180,E1 -17764.675,E2 -17764.675} C_VEL
LIN {X 0,Y 271.901,Z 433.647,A -85,B 0,C 180,E1 -17766.748,E2 -17766.748} C_VEL
LIN {X 0,Y 271.746,Z 431.04,A -85,B 0,C 180,E1 -17769.116,E2 -17769.116} C_VEL
LIN {X 0,Y 271.174,Z 427.645,A -85,B 0,C 180,E1 -17772.364,E2 -17772.364} C_VEL
LIN {X 0,Y 270.461,Z 423.417,A -85,B 0,C 180,E1 -17776.684,E2 -17776.684} C_VEL
LIN {X 0,Y 270.184,Z 421.832,A -85,B 0,C 180,E1 -17778.483,E2 -17778.483} C_VEL
LIN {X 0,Y 270.207,Z 421.831,A -85,B 0,C 180,E1 -17781.374,E2 -17781.374} C_VEL
LIN {X 0,Y 270.203,Z 421.832,A -85,B 0,C 180,E1 -17785.095,E2 -17785.095} C_VEL
LIN {X 0,Y 270.201,Z 421.829,A -85,B 0,C 180,E1 -17789.131,E2 -17789.131} C_VEL
LIN {X 0,Y 270.264,Z 421.819,A -85,B 0,C 180,E1 -17792.146,E2 -17792.146} C_VEL
LIN {X 0,Y 270.278,Z 421.817,A -85,B 0,C 180,E1 -17795.519,E2 -17795.519} C_VEL
LIN {X 0,Y 270.303,Z 421.816,A -85,B 0,C 180,E1 -17800.245,E2 -17800.245} C_VEL
LIN {X 0,Y 270.405,Z 421.802,A -85,B 0,C 180,E1 -17804.935,E2 -17804.935} C_VEL
LIN {X 0,Y 270.444,Z 421.796,A -85,B 0,C 180,E1 -17809.519,E2 -17809.519} C_VEL
LIN {X 0,Y 270.613,Z 421.776,A -85,B 0,C 180,E1 -17812.539,E2 -17812.539} C_VEL
LIN {X 0,Y 270.789,Z 421.755,A -85,B 0,C 180,E1 -17818.513,E2 -17818.513} C_VEL
LIN {X 0,Y 270.789,Z 421.753,A -85,B 0,C 180,E1 -17821.487,E2 -17821.487} C_VEL
LIN {X 0,Y 270.613,Z 421.775,A -85,B 0,C 180,E1 -17827.461,E2 -17827.461} C_VEL
LIN {X 0,Y 270.444,Z 421.796,A -85,B 0,C 180,E1 -17830.481,E2 -17830.481} C_VEL
LIN {X 0,Y 270.405,Z 421.8,A -85,B 0,C 180,E1 -17835.065,E2 -17835.065} C_VEL
LIN {X 0,Y 270.303,Z 421.813,A -85,B 0,C 180,E1 -17839.756,E2 -17839.756} C_VEL
LIN {X 0,Y 270.275,Z 421.816,A -85,B 0,C 180,E1 -17844.586,E2 -17844.586} C_VEL
LIN {X 0,Y 270.271,Z 421.819,A -85,B 0,C 180,E1 -17847.909,E2 -17847.909} C_VEL
LIN {X 0,Y 270.186,Z 421.829,A -85,B 0,C 180,E1 -17851.348,E2 -17851.348} C_VEL
LIN {X 0,Y 270.216,Z 421.824,A -85,B 0,C 180,E1 -17854.904,E2 -17854.904} C_VEL
LIN {X 0,Y 270.223,Z 421.824,A -85,B 0,C 180,E1 -17858.717,E2 -17858.717} C_VEL
LIN {X 0,Y 270.173,Z 421.832,A -85,B 0,C 180,E1 -17863.251,E2 -17863.251} C_VEL
LIN {X 0,Y 270.176,Z 421.833,A -85,B 0,C 180,E1 -17867.443,E2 -17867.443} C_VEL
LIN {X 0,Y 270.175,Z 421.832,A -85,B 0,C 180,E1 -17869.434,E2 -17869.434} C_VEL
LIN {X 0,Y 270.246,Z 422.283,A -85,B 0,C 180,E1 -17871.381,E2 -17871.381} C_VEL
LIN {X 0,Y 270.277,Z 425.288,A -85,B 0,C 180,E1 -17875.106,E2 -17875.106} C_VEL
LIN {X 0,Y 270.011,Z 428.828,A -85,B 0,C 180,E1 -17879.199,E2 -17879.199} C_VEL
LIN {X 0,Y 269.689,Z 432.042,A -85,B 0,C 180,E1 -17882.716,E2 -17882.716} C_VEL
LIN {X 0,Y 274.137,Z 446.272,A -85,B 0,C 180,E1 -17883.976,E2 -17883.976} C_VEL
LIN {X 0,Y 276.928,Z 457.342,A -85,B 0,C 180,E1 -17885.132,E2 -17885.132} C_VEL
LIN {X 0,Y 279.052,Z 468.802,A -85,B 0,C 180,E1 -17886.514,E2 -17886.514} C_VEL
LIN {X 0,Y 279.734,Z 474.585,A -85,B 0,C 180,E1 -17887.289,E2 -17887.289} C_VEL
LIN {X 0,Y 277.902,Z 486.316,A -85,B 0,C 180,E1 -17888.877,E2 -17888.877} C_VEL
LIN {X 0,Y 276.18,Z 496.794,A -85,B 0,C 180,E1 -17890.682,E2 -17890.682} C_VEL
LIN {X 0,Y 274.418,Z 505.28,A -85,B 0,C 180,E1 -17892.487,E2 -17892.487} C_VEL
LIN {X 0,Y 272.623,Z 513.528,A -85,B 0,C 180,E1 -17894.679,E2 -17894.679} C_VEL
LIN {X 0,Y 271.423,Z 519.167,A -85,B 0,C 180,E1 -17896.524,E2 -17896.524} C_VEL
LIN {X 0,Y 270.207,Z 524.664,A -85,B 0,C 180,E1 -17898.751,E2 -17898.751} C_VEL
LIN {X 0,Y 269.35,Z 528.976,A -85,B 0,C 180,E1 -17900.993,E2 -17900.993} C_VEL
LIN {X 0,Y 268.751,Z 532.622,A -85,B 0,C 180,E1 -17903.58,E2 -17903.58} C_VEL
LIN {X 0,Y 268.486,Z 534.501,A -85,B 0,C 180,E1 -17905.496,E2 -17905.496} C_VEL
LIN {X 0,Y 268.362,Z 535.491,A -85,B 0,C 180,E1 -17906.998,E2 -17906.998} C_VEL
LIN {X 0,Y 268.21,Z 536.332,A -85,B 0,C 180,E1 -17910,E2 -17910} C_VEL
LIN {X 0,Y 268.234,Z 536.139,A -85,B 0,C 180,E1 -17911.502,E2 -17911.502} C_VEL
LIN {X 0,Y 268.36,Z 535.552,A -85,B 0,C 180,E1 -17913.003,E2 -17913.003} C_VEL
LIN {X 0,Y 268.481,Z 534.585,A -85,B 0,C 180,E1 -17914.504,E2 -17914.504} C_VEL
LIN {X 0,Y 268.791,Z 532.667,A -85,B 0,C 180,E1 -17916.495,E2 -17916.495} C_VEL
LIN {X 0,Y 269.348,Z 529.168,A -85,B 0,C 180,E1 -17919.007,E2 -17919.007} C_VEL
LIN {X 0,Y 270.18,Z 524.916,A -85,B 0,C 180,E1 -17921.25,E2 -17921.25} C_VEL
LIN {X 0,Y 271.59,Z 518.474,A -85,B 0,C 180,E1 -17923.849,E2 -17923.849} C_VEL
LIN {X 0,Y 273.094,Z 511.393,A -85,B 0,C 180,E1 -17926.06,E2 -17926.06} C_VEL
LIN {X 0,Y 275.057,Z 502.567,A -85,B 0,C 180,E1 -17928.24,E2 -17928.24} C_VEL
LIN {X 0,Y 276.689,Z 493.363,A -85,B 0,C 180,E1 -17930.085,E2 -17930.085} C_VEL
LIN {X 0,Y 278.437,Z 483.48,A -85,B 0,C 180,E1 -17931.663,E2 -17931.663} C_VEL
LIN {X 0,Y 279.75,Z 475.377,A -85,B 0,C 180,E1 -17932.722,E2 -17932.722} C_VEL
LIN {X 0,Y 278.426,Z 464.662,A -85,B 0,C 180,E1 -17934.131,E2 -17934.131} C_VEL
LIN {X 0,Y 275.879,Z 452.665,A -85,B 0,C 180,E1 -17935.498,E2 -17935.498} C_VEL
LIN {X 0,Y 272.348,Z 440.202,A -85,B 0,C 180,E1 -17936.712,E2 -17936.712} C_VEL
LIN {X 0,Y 269.704,Z 432.043,A -85,B 0,C 180,E1 -17937.411,E2 -17937.411} C_VEL
LIN {X 0,Y 270.023,Z 428.44,A -85,B 0,C 180,E1 -17941.369,E2 -17941.369} C_VEL
LIN {X 0,Y 270.298,Z 425.428,A -85,B 0,C 180,E1 -17944.892,E2 -17944.892} C_VEL
LIN {X 0,Y 270.255,Z 422.31,A -85,B 0,C 180,E1 -17948.725,E2 -17948.725} C_VEL
LIN {X 0,Y 270.171,Z 421.83,A -85,B 0,C 180,E1 -17951.028,E2 -17951.028} C_VEL
LIN {X 0,Y 270.168,Z 421.83,A -85,B 0,C 180,E1 -17955.383,E2 -17955.383} C_VEL
LIN {X 0,Y 270.177,Z 421.829,A -85,B 0,C 180,E1 -17959.434,E2 -17959.434} C_VEL
LIN {X 0,Y 270.257,Z 421.819,A -85,B 0,C 180,E1 -17963.722,E2 -17963.722} C_VEL
LIN {X 0,Y 270.207,Z 421.826,A -85,B 0,C 180,E1 -17966.893,E2 -17966.893} C_VEL
LIN {X 0,Y 270.199,Z 421.827,A -85,B 0,C 180,E1 -17970.383,E2 -17970.383} C_VEL
LIN {X 0,Y 270.265,Z 421.818,A -85,B 0,C 180,E1 -17973.764,E2 -17973.764} C_VEL
LIN {X 0,Y 270.239,Z 421.821,A -85,B 0,C 180,E1 -17977.039,E2 -17977.039} C_VEL
LIN {X 0,Y 270.305,Z 421.816,A -85,B 0,C 180,E1 -17980.245,E2 -17980.245} C_VEL
LIN {X 0,Y 270.406,Z 421.799,A -85,B 0,C 180,E1 -17984.935,E2 -17984.935} C_VEL
LIN {X 0,Y 270.445,Z 421.796,A -85,B 0,C 180,E1 -17989.519,E2 -17989.519} C_VEL
LIN {X 0,Y 270.614,Z 421.775,A -85,B 0,C 180,E1 -17992.539,E2 -17992.539} C_VEL
LIN {X 0,Y 270.789,Z 421.753,A -85,B 0,C 180,E1 -17998.513,E2 -17998.513} C_VEL
LIN {X 0,Y 270.79,Z 421.755,A -85,B 0,C 180,E1 -18001.487,E2 -18001.487} C_VEL
LIN {X 0,Y 270.614,Z 421.778,A -85,B 0,C 180,E1 -18007.461,E2 -18007.461} C_VEL
LIN {X 0,Y 270.445,Z 421.794,A -85,B 0,C 180,E1 -18010.481,E2 -18010.481} C_VEL
LIN {X 0,Y 270.406,Z 421.802,A -85,B 0,C 180,E1 -18015.064,E2 -18015.064} C_VEL
LIN {X 0,Y 270.372,Z 421.805,A -85,B 0,C 180,E1 -18016.101,E2 -18016.101} C_VEL
LIN {X 0,Y 269.651,Z 421.898,A -85,B 0,C 180,E1 -18017.345,E2 -18017.345} C_VEL
LIN {X 0,Y 266.72,Z 422.264,A -85,B 0,C 180,E1 -18019.369,E2 -18019.369} C_VEL
LIN {X 0,Y 264.263,Z 422.567,A -85,B 0,C 180,E1 -18021.016,E2 -18021.016} C_VEL
LIN {X 0,Y 263.223,Z 422.695,A -85,B 0,C 180,E1 -18022.294,E2 -18022.294} C_VEL
LIN {X 0,Y 263.145,Z 422.702,A -85,B 0,C 180,E1 -18022.727,E2 -18022.727} C_VEL
LIN {X 0,Y 263.21,Z 422.701,A -85,B 0,C 180,E1 -18025.291,E2 -18025.291} C_VEL
LIN {X 0,Y 263.167,Z 422.701,A -85,B 0,C 180,E1 -18028.731,E2 -18028.731} C_VEL
LIN {X 0,Y 263.134,Z 422.699,A -85,B 0,C 180,E1 -18032.288,E2 -18032.288} C_VEL
LIN {X 0,Y 263.185,Z 422.702,A -85,B 0,C 180,E1 -18036.763,E2 -18036.763} C_VEL
LIN {X 0,Y 263.162,Z 422.89,A -85,B 0,C 180,E1 -18041.191,E2 -18041.191} C_VEL
LIN {X 0,Y 263.612,Z 425.388,A -85,B 0,C 180,E1 -18043.959,E2 -18043.959} C_VEL
LIN {X 0,Y 264.287,Z 429.608,A -85,B 0,C 180,E1 -18048.332,E2 -18048.332} C_VEL
LIN {X 0,Y 264.763,Z 432.762,A -85,B 0,C 180,E1 -18051.406,E2 -18051.406} C_VEL
LIN {X 0,Y 264.842,Z 435.898,A -85,B 0,C 180,E1 -18054.281,E2 -18054.281} C_VEL
LIN {X 0,Y 264.135,Z 440.046,A -85,B 0,C 180,E1 -18057.849,E2 -18057.849} C_VEL
LIN {X 0,Y 263.287,Z 444.867,A -85,B 0,C 180,E1 -18061.899,E2 -18061.899} C_VEL
LIN {X 0,Y 264.844,Z 450.771,A -85,B 0,C 180,E1 -18062.34,E2 -18062.34} C_VEL
LIN {X 0,Y 267.781,Z 462.831,A -85,B 0,C 180,E1 -18063.408,E2 -18063.408} C_VEL
LIN {X 0,Y 269.854,Z 474.617,A -85,B 0,C 180,E1 -18064.643,E2 -18064.643} C_VEL
LIN {X 0,Y 271.08,Z 486.689,A -85,B 0,C 180,E1 -18066.128,E2 -18066.128} C_VEL
LIN {X 0,Y 271.346,Z 495.236,A -85,B 0,C 180,E1 -18067.339,E2 -18067.339} C_VEL
LIN {X 0,Y 269.443,Z 505.885,A -85,B 0,C 180,E1 -18068.983,E2 -18068.983} C_VEL
LIN {X 0,Y 267.57,Z 515.488,A -85,B 0,C 180,E1 -18070.833,E2 -18070.833} C_VEL
LIN {X 0,Y 265.959,Z 523.354,A -85,B 0,C 180,E1 -18072.705,E2 -18072.705} C_VEL
LIN {X 0,Y 264.26,Z 531.038,A -85,B 0,C 180,E1 -18074.971,E2 -18074.971} C_VEL
LIN {X 0,Y 262.719,Z 538.129,A -85,B 0,C 180,E1 -18077.642,E2 -18077.642} C_VEL
LIN {X 0,Y 261.909,Z 542.852,A -85,B 0,C 180,E1 -18079.955,E2 -18079.955} C_VEL
LIN {X 0,Y 261.356,Z 546.461,A -85,B 0,C 180,E1 -18082.273,E2 -18082.273} C_VEL
LIN {X 0,Y 261.085,Z 549.319,A -85,B 0,C 180,E1 -18084.864,E2 -18084.864} C_VEL
LIN {X 0,Y 261.064,Z 550.722,A -85,B 0,C 180,E1 -18086.913,E2 -18086.913} C_VEL
LIN {X 0,Y 261.116,Z 551.332,A -85,B 0,C 180,E1 -18088.458,E2 -18088.458} C_VEL
LIN {X 0,Y 261.128,Z 551.546,A -85,B 0,C 180,E1 -18090,E2 -18090} C_VEL
LIN {X 0,Y 261.116,Z 551.324,A -85,B 0,C 180,E1 -18091.542,E2 -18091.542} C_VEL
LIN {X 0,Y 261.063,Z 550.708,A -85,B 0,C 180,E1 -18093.086,E2 -18093.086} C_VEL
LIN {X 0,Y 261.085,Z 549.293,A -85,B 0,C 180,E1 -18095.137,E2 -18095.137} C_VEL
LIN {X 0,Y 261.356,Z 546.424,A -85,B 0,C 180,E1 -18097.727,E2 -18097.727} C_VEL
LIN {X 0,Y 261.909,Z 542.797,A -85,B 0,C 180,E1 -18100.045,E2 -18100.045} C_VEL
LIN {X 0,Y 262.719,Z 538.059,A -85,B 0,C 180,E1 -18102.357,E2 -18102.357} C_VEL
LIN {X 0,Y 264.26,Z 530.953,A -85,B 0,C 180,E1 -18105.029,E2 -18105.029} C_VEL
LIN {X 0,Y 265.959,Z 523.24,A -85,B 0,C 180,E1 -18107.294,E2 -18107.294} C_VEL
LIN {X 0,Y 267.481,Z 515.651,A -85,B 0,C 180,E1 -18109.105,E2 -18109.105} C_VEL
LIN {X 0,Y 269.431,Z 505.715,A -85,B 0,C 180,E1 -18111.018,E2 -18111.018} C_VEL
LIN {X 0,Y 271.231,Z 496.33,A -85,B 0,C 180,E1 -18112.47,E2 -18112.47} C_VEL
LIN {X 0,Y 271.077,Z 487.845,A -85,B 0,C 180,E1 -18113.692,E2 -18113.692} C_VEL
LIN {X 0,Y 270.09,Z 476.632,A -85,B 0,C 180,E1 -18115.092,E2 -18115.092} C_VEL
LIN {X 0,Y 268.167,Z 464.624,A -85,B 0,C 180,E1 -18116.373,E2 -18116.373} C_VEL
LIN {X 0,Y 265.059,Z 451.704,A -85,B 0,C 180,E1 -18117.553,E2 -18117.553} C_VEL
LIN {X 0,Y 263.289,Z 444.793,A -85,B 0,C 180,E1 -18118.117,E2 -18118.117} C_VEL
LIN {X 0,Y 264.199,Z 440.003,A -85,B 0,C 180,E1 -18122.142,E2 -18122.142} C_VEL
LIN {X 0,Y 264.818,Z 435.839,A -85,B 0,C 180,E1 -18125.722,E2 -18125.722} C_VEL
LIN {X 0,Y 264.764,Z 432.698,A -85,B 0,C 180,E1 -18128.594,E2 -18128.594} C_VEL
LIN {X 0,Y 264.281,Z 429.346,A -85,B 0,C 180,E1 -18131.875,E2 -18131.875} C_VEL
LIN {X 0,Y 263.561,Z 425.281,A -85,B 0,C 180,E1 -18136.108,E2 -18136.108} C_VEL
LIN {X 0,Y 263.13,Z 422.711,A -85,B 0,C 180,E1 -18139.035,E2 -18139.035} C_VEL
LIN {X 0,Y 263.184,Z 422.706,A -85,B 0,C 180,E1 -18143.236,E2 -18143.236} C_VEL
LIN {X 0,Y 263.133,Z 422.709,A -85,B 0,C 180,E1 -18147.712,E2 -18147.712} C_VEL
LIN {X 0,Y 263.196,Z 422.699,A -85,B 0,C 180,E1 -18151.785,E2 -18151.785} C_VEL
LIN {X 0,Y 263.227,Z 422.696,A -85,B 0,C 180,E1 -18155.2,E2 -18155.2} C_VEL
LIN {X 0,Y 263.265,Z 422.691,A -85,B 0,C 180,E1 -18159.693,E2 -18159.693} C_VEL
LIN {X 0,Y 263.352,Z 422.682,A -85,B 0,C 180,E1 -18164.522,E2 -18164.522} C_VEL
LIN {X 0,Y 263.376,Z 422.676,A -85,B 0,C 180,E1 -18169.235,E2 -18169.235} C_VEL
LIN {X 0,Y 263.574,Z 422.654,A -85,B 0,C 180,E1 -18172.339,E2 -18172.339} C_VEL
LIN {X 0,Y 263.753,Z 422.632,A -85,B 0,C 180,E1 -18178.473,E2 -18178.473} C_VEL
LIN {X 0,Y 263.753,Z 422.63,A -85,B 0,C 180,E1 -18181.527,E2 -18181.527} C_VEL
LIN {X 0,Y 263.575,Z 422.653,A -85,B 0,C 180,E1 -18187.662,E2 -18187.662} C_VEL
LIN {X 0,Y 263.376,Z 422.675,A -85,B 0,C 180,E1 -18190.766,E2 -18190.766} C_VEL
LIN {X 0,Y 263.352,Z 422.68,A -85,B 0,C 180,E1 -18195.478,E2 -18195.478} C_VEL
LIN {X 0,Y 263.265,Z 422.69,A -85,B 0,C 180,E1 -18200.307,E2 -18200.307} C_VEL
LIN {X 0,Y 263.209,Z 422.698,A -85,B 0,C 180,E1 -18205.291,E2 -18205.291} C_VEL
LIN {X 0,Y 263.177,Z 422.7,A -85,B 0,C 180,E1 -18208.73,E2 -18208.73} C_VEL
LIN {X 0,Y 263.135,Z 422.706,A -85,B 0,C 180,E1 -18212.288,E2 -18212.288} C_VEL
LIN {X 0,Y 263.189,Z 422.701,A -85,B 0,C 180,E1 -18215.978,E2 -18215.978} C_VEL
LIN {X 0,Y 263.116,Z 422.71,A -85,B 0,C 180,E1 -18219.871,E2 -18219.871} C_VEL
LIN {X 0,Y 263.129,Z 422.709,A -85,B 0,C 180,E1 -18223.983,E2 -18223.983} C_VEL
LIN {X 0,Y 263.126,Z 422.71,A -85,B 0,C 180,E1 -18228.407,E2 -18228.407} C_VEL
LIN {X 0,Y 263.135,Z 422.966,A -85,B 0,C 180,E1 -18230.765,E2 -18230.765} C_VEL
LIN {X 0,Y 263.286,Z 425.501,A -85,B 0,C 180,E1 -18234.038,E2 -18234.038} C_VEL
LIN {X 0,Y 263.068,Z 428.532,A -85,B 0,C 180,E1 -18237.703,E2 -18237.703} C_VEL
LIN {X 0,Y 262.693,Z 432.264,A -85,B 0,C 180,E1 -18241.919,E2 -18241.919} C_VEL
LIN {X 0,Y 264.597,Z 437.959,A -85,B 0,C 180,E1 -18242.427,E2 -18242.427} C_VEL
LIN {X 0,Y 268.038,Z 449.21,A -85,B 0,C 180,E1 -18243.529,E2 -18243.529} C_VEL
LIN {X 0,Y 270.615,Z 460.014,A -85,B 0,C 180,E1 -18244.741,E2 -18244.741} C_VEL
LIN {X 0,Y 272.496,Z 470.843,A -85,B 0,C 180,E1 -18246.139,E2 -18246.139} C_VEL
LIN {X 0,Y 273.043,Z 476.379,A -85,B 0,C 180,E1 -18246.923,E2 -18246.923} C_VEL
LIN {X 0,Y 271.113,Z 487.693,A -85,B 0,C 180,E1 -18248.521,E2 -18248.521} C_VEL
LIN {X 0,Y 269.502,Z 497.001,A -85,B 0,C 180,E1 -18250.184,E2 -18250.184} C_VEL
LIN {X 0,Y 267.663,Z 505.487,A -85,B 0,C 180,E1 -18252.03,E2 -18252.03} C_VEL
LIN {X 0,Y 265.789,Z 513.734,A -85,B 0,C 180,E1 -18254.274,E2 -18254.274} C_VEL
LIN {X 0,Y 264.518,Z 519.373,A -85,B 0,C 180,E1 -18256.165,E2 -18256.165} C_VEL
LIN {X 0,Y 263.249,Z 524.869,A -85,B 0,C 180,E1 -18258.45,E2 -18258.45} C_VEL
LIN {X 0,Y 262.326,Z 529.181,A -85,B 0,C 180,E1 -18260.75,E2 -18260.75} C_VEL
LIN {X 0,Y 261.633,Z 533.13,A -85,B 0,C 180,E1 -18263.67,E2 -18263.67} C_VEL
LIN {X 0,Y 261.4,Z 534.706,A -85,B 0,C 180,E1 -18265.374,E2 -18265.374} C_VEL
LIN {X 0,Y 261.277,Z 535.696,A -85,B 0,C 180,E1 -18266.916,E2 -18266.916} C_VEL
LIN {X 0,Y 261.136,Z 536.535,A -85,B 0,C 180,E1 -18270,E2 -18270} C_VEL
LIN {X 0,Y 261.164,Z 536.342,A -85,B 0,C 180,E1 -18271.542,E2 -18271.542} C_VEL
LIN {X 0,Y 261.275,Z 535.755,A -85,B 0,C 180,E1 -18273.084,E2 -18273.084} C_VEL
LIN {X 0,Y 261.621,Z 533.432,A -85,B 0,C 180,E1 -18276.169,E2 -18276.169} C_VEL
LIN {X 0,Y 262.115,Z 530.566,A -85,B 0,C 180,E1 -18278.48,E2 -18278.48} C_VEL
LIN {X 0,Y 262.873,Z 526.678,A -85,B 0,C 180,E1 -18280.787,E2 -18280.787} C_VEL
LIN {X 0,Y 264.007,Z 521.658,A -85,B 0,C 180,E1 -18283.078,E2 -18283.078} C_VEL
LIN {X 0,Y 265.377,Z 515.338,A -85,B 0,C 180,E1 -18285.357,E2 -18285.357} C_VEL
LIN {X 0,Y 267.251,Z 507.422,A -85,B 0,C 180,E1 -18287.603,E2 -18287.603} C_VEL
LIN {X 0,Y 268.983,Z 499.353,A -85,B 0,C 180,E1 -18289.459,E2 -18289.459} C_VEL
LIN {X 0,Y 270.782,Z 489.509,A -85,B 0,C 180,E1 -18291.307,E2 -18291.307} C_VEL
LIN {X 0,Y 272.798,Z 478.466,A -85,B 0,C 180,E1 -18292.927,E2 -18292.927} C_VEL
LIN {X 0,Y 272.933,Z 474.316,A -85,B 0,C 180,E1 -18293.497,E2 -18293.497} C_VEL
LIN {X 0,Y 271.336,Z 463.329,A -85,B 0,C 180,E1 -18294.966,E2 -18294.966} C_VEL
LIN {X 0,Y 268.642,Z 451.336,A -85,B 0,C 180,E1 -18296.361,E2 -18296.361} C_VEL
LIN {X 0,Y 264.941,Z 438.75,A -85,B 0,C 180,E1 -18297.619,E2 -18297.619} C_VEL
LIN {X 0,Y 262.77,Z 432.775,A -85,B 0,C 180,E1 -18298.159,E2 -18298.159} C_VEL
LIN {X 0,Y 262.702,Z 432.231,A -85,B 0,C 180,E1 -18298.25,E2 -18298.25} C_VEL
LIN {X 0,Y 263.058,Z 428.648,A -85,B 0,C 180,E1 -18302.299,E2 -18302.299} C_VEL
LIN {X 0,Y 263.253,Z 427.1,A -85,B 0,C 180,E1 -18304.146,E2 -18304.146} C_VEL
LIN {X 0,Y 263.241,Z 424.099,A -85,B 0,C 180,E1 -18307.883,E2 -18307.883} C_VEL
LIN {X 0,Y 263.124,Z 422.708,A -85,B 0,C 180,E1 -18309.869,E2 -18309.869} C_VEL
LIN {X 0,Y 263.13,Z 422.706,A -85,B 0,C 180,E1 -18313.983,E2 -18313.983} C_VEL
LIN {X 0,Y 263.127,Z 422.71,A -85,B 0,C 180,E1 -18318.406,E2 -18318.406} C_VEL
LIN {X 0,Y 263.168,Z 422.702,A -85,B 0,C 180,E1 -18322.104,E2 -18322.104} C_VEL
LIN {X 0,Y 263.186,Z 422.701,A -85,B 0,C 180,E1 -18325.89,E2 -18325.89} C_VEL
LIN {X 0,Y 263.143,Z 422.705,A -85,B 0,C 180,E1 -18329.506,E2 -18329.506} C_VEL
LIN {X 0,Y 263.194,Z 422.698,A -85,B 0,C 180,E1 -18333.003,E2 -18333.003} C_VEL
LIN {X 0,Y 263.189,Z 422.703,A -85,B 0,C 180,E1 -18336.387,E2 -18336.387} C_VEL
LIN {X 0,Y 263.267,Z 422.69,A -85,B 0,C 180,E1 -18339.694,E2 -18339.694} C_VEL
LIN {X 0,Y 263.354,Z 422.679,A -85,B 0,C 180,E1 -18344.522,E2 -18344.522} C_VEL
LIN {X 0,Y 263.377,Z 422.676,A -85,B 0,C 180,E1 -18349.234,E2 -18349.234} C_VEL
LIN {X 0,Y 263.576,Z 422.653,A -85,B 0,C 180,E1 -18352.338,E2 -18352.338} C_VEL
LIN {X 0,Y 263.753,Z 422.629,A -85,B 0,C 180,E1 -18358.473,E2 -18358.473} C_VEL
LIN {X 0,Y 263.754,Z 422.632,A -85,B 0,C 180,E1 -18361.527,E2 -18361.527} C_VEL
LIN {X 0,Y 263.576,Z 422.654,A -85,B 0,C 180,E1 -18367.661,E2 -18367.661} C_VEL
LIN {X 0,Y 263.377,Z 422.675,A -85,B 0,C 180,E1 -18370.765,E2 -18370.765} C_VEL
LIN {X 0,Y 263.354,Z 422.682,A -85,B 0,C 180,E1 -18375.478,E2 -18375.478} C_VEL
LIN {X 0,Y 263.266,Z 422.689,A -85,B 0,C 180,E1 -18380.306,E2 -18380.306} C_VEL
LIN {X 0,Y 263.145,Z 422.702,A -85,B 0,C 180,E1 -18382.727,E2 -18382.727} C_VEL
LIN {X 0,Y 262.491,Z 422.787,A -85,B 0,C 180,E1 -18384.004,E2 -18384.004} C_VEL
LIN {X 0,Y 259.636,Z 423.142,A -85,B 0,C 180,E1 -18386.085,E2 -18386.085} C_VEL
LIN {X 0,Y 257.211,Z 423.443,A -85,B 0,C 180,E1 -18387.778,E2 -18387.778} C_VEL
LIN {X 0,Y 256.181,Z 423.572,A -85,B 0,C 180,E1 -18389.091,E2 -18389.091} C_VEL
LIN {X 0,Y 256.104,Z 423.584,A -85,B 0,C 180,E1 -18389.535,E2 -18389.535} C_VEL
LIN {X 0,Y 256.069,Z 423.578,A -85,B 0,C 180,E1 -18393.293,E2 -18393.293} C_VEL
LIN {X 0,Y 256.117,Z 423.584,A -85,B 0,C 180,E1 -18397.271,E2 -18397.271} C_VEL
LIN {X 0,Y 256.082,Z 423.605,A -85,B 0,C 180,E1 -18400.419,E2 -18400.419} C_VEL
LIN {X 0,Y 256.714,Z 427.289,A -85,B 0,C 180,E1 -18404.618,E2 -18404.618} C_VEL
LIN {X 0,Y 257.407,Z 431.509,A -85,B 0,C 180,E1 -18409.059,E2 -18409.059} C_VEL
LIN {X 0,Y 257.797,Z 434.736,A -85,B 0,C 180,E1 -18412.241,E2 -18412.241} C_VEL
LIN {X 0,Y 257.692,Z 437.769,A -85,B 0,C 180,E1 -18415.059,E2 -18415.059} C_VEL
LIN {X 0,Y 256.699,Z 442.921,A -85,B 0,C 180,E1 -18419.569,E2 -18419.569} C_VEL
LIN {X 0,Y 256.402,Z 444.663,A -85,B 0,C 180,E1 -18421.069,E2 -18421.069} C_VEL
LIN {X 0,Y 259.859,Z 457.788,A -85,B 0,C 180,E1 -18422.187,E2 -18422.187} C_VEL
LIN {X 0,Y 262.434,Z 470.248,A -85,B 0,C 180,E1 -18423.471,E2 -18423.471} C_VEL
LIN {X 0,Y 263.943,Z 481.911,A -85,B 0,C 180,E1 -18424.866,E2 -18424.866} C_VEL
LIN {X 0,Y 264.614,Z 492.677,A -85,B 0,C 180,E1 -18426.371,E2 -18426.371} C_VEL
LIN {X 0,Y 264.443,Z 497.628,A -85,B 0,C 180,E1 -18427.127,E2 -18427.127} C_VEL
LIN {X 0,Y 262.337,Z 507.793,A -85,B 0,C 180,E1 -18428.797,E2 -18428.797} C_VEL
LIN {X 0,Y 260.268,Z 517.928,A -85,B 0,C 180,E1 -18430.927,E2 -18430.927} C_VEL
LIN {X 0,Y 258.492,Z 525.885,A -85,B 0,C 180,E1 -18433.006,E2 -18433.006} C_VEL
LIN {X 0,Y 256.871,Z 533.073,A -85,B 0,C 180,E1 -18435.34,E2 -18435.34} C_VEL
LIN {X 0,Y 255.745,Z 537.925,A -85,B 0,C 180,E1 -18437.3,E2 -18437.3} C_VEL
LIN {X 0,Y 254.876,Z 542.648,A -85,B 0,C 180,E1 -18439.675,E2 -18439.675} C_VEL
LIN {X 0,Y 254.316,Z 546.258,A -85,B 0,C 180,E1 -18442.058,E2 -18442.058} C_VEL
LIN {X 0,Y 253.99,Z 549.319,A -85,B 0,C 180,E1 -18444.961,E2 -18444.961} C_VEL
LIN {X 0,Y 253.963,Z 550.518,A -85,B 0,C 180,E1 -18446.827,E2 -18446.827} C_VEL
LIN {X 0,Y 254.021,Z 551.128,A -85,B 0,C 180,E1 -18448.414,E2 -18448.414} C_VEL
LIN {X 0,Y 254.056,Z 551.343,A -85,B 0,C 180,E1 -18450,E2 -18450} C_VEL
LIN {X 0,Y 254.021,Z 551.12,A -85,B 0,C 180,E1 -18451.585,E2 -18451.585} C_VEL
LIN {X 0,Y 253.962,Z 550.504,A -85,B 0,C 180,E1 -18453.173,E2 -18453.173} C_VEL
LIN {X 0,Y 253.99,Z 549.299,A -85,B 0,C 180,E1 -18455.039,E2 -18455.039} C_VEL
LIN {X 0,Y 254.315,Z 546.219,A -85,B 0,C 180,E1 -18457.942,E2 -18457.942} C_VEL
LIN {X 0,Y 254.876,Z 542.59,A -85,B 0,C 180,E1 -18460.325,E2 -18460.325} C_VEL
LIN {X 0,Y 255.744,Z 537.852,A -85,B 0,C 180,E1 -18462.7,E2 -18462.7} C_VEL
LIN {X 0,Y 257.401,Z 530.747,A -85,B 0,C 180,E1 -18465.439,E2 -18465.439} C_VEL
LIN {X 0,Y 259.182,Z 523.033,A -85,B 0,C 180,E1 -18467.761,E2 -18467.761} C_VEL
LIN {X 0,Y 261.164,Z 513.35,A -85,B 0,C 180,E1 -18470.066,E2 -18470.066} C_VEL
LIN {X 0,Y 263.25,Z 503.362,A -85,B 0,C 180,E1 -18471.948,E2 -18471.948} C_VEL
LIN {X 0,Y 264.601,Z 496.119,A -85,B 0,C 180,E1 -18473.065,E2 -18473.065} C_VEL
LIN {X 0,Y 264.132,Z 484.846,A -85,B 0,C 180,E1 -18474.72,E2 -18474.72} C_VEL
LIN {X 0,Y 262.871,Z 473.178,A -85,B 0,C 180,E1 -18476.169,E2 -18476.169} C_VEL
LIN {X 0,Y 260.508,Z 460.57,A -85,B 0,C 180,E1 -18477.502,E2 -18477.502} C_VEL
LIN {X 0,Y 257.038,Z 447.385,A -85,B 0,C 180,E1 -18478.688,E2 -18478.688} C_VEL
LIN {X 0,Y 256.408,Z 444.612,A -85,B 0,C 180,E1 -18478.909,E2 -18478.909} C_VEL
LIN {X 0,Y 257.313,Z 439.794,A -85,B 0,C 180,E1 -18483.111,E2 -18483.111} C_VEL
LIN {X 0,Y 257.73,Z 437.534,A -85,B 0,C 180,E1 -18485.108,E2 -18485.108} C_VEL
LIN {X 0,Y 257.785,Z 434.665,A -85,B 0,C 180,E1 -18487.756,E2 -18487.756} C_VEL
LIN {X 0,Y 257.419,Z 431.442,A -85,B 0,C 180,E1 -18490.938,E2 -18490.938} C_VEL
LIN {X 0,Y 256.681,Z 427.238,A -85,B 0,C 180,E1 -18495.389,E2 -18495.389} C_VEL
LIN {X 0,Y 256.091,Z 423.588,A -85,B 0,C 180,E1 -18499.583,E2 -18499.583} C_VEL
LIN {X 0,Y 256.132,Z 423.585,A -85,B 0,C 180,E1 -18502.868,E2 -18502.868} C_VEL
LIN {X 0,Y 256.068,Z 423.592,A -85,B 0,C 180,E1 -18506.707,E2 -18506.707} C_VEL
LIN {X 0,Y 256.104,Z 423.585,A -85,B 0,C 180,E1 -18510.399,E2 -18510.399} C_VEL
LIN {X 0,Y 256.189,Z 423.574,A -85,B 0,C 180,E1 -18514.862,E2 -18514.862} C_VEL
LIN {X 0,Y 256.168,Z 423.576,A -85,B 0,C 180,E1 -18519.105,E2 -18519.105} C_VEL
LIN {X 0,Y 256.301,Z 423.56,A -85,B 0,C 180,E1 -18524.085,E2 -18524.085} C_VEL
LIN {X 0,Y 256.312,Z 423.557,A -85,B 0,C 180,E1 -18528.934,E2 -18528.934} C_VEL
LIN {X 0,Y 256.542,Z 423.53,A -85,B 0,C 180,E1 -18532.127,E2 -18532.127} C_VEL
LIN {X 0,Y 256.716,Z 423.509,A -85,B 0,C 180,E1 -18538.431,E2 -18538.431} C_VEL
LIN {X 0,Y 256.716,Z 423.506,A -85,B 0,C 180,E1 -18541.569,E2 -18541.569} C_VEL
LIN {X 0,Y 256.542,Z 423.53,A -85,B 0,C 180,E1 -18547.873,E2 -18547.873} C_VEL
LIN {X 0,Y 256.312,Z 423.555,A -85,B 0,C 180,E1 -18551.066,E2 -18551.066} C_VEL
LIN {X 0,Y 256.301,Z 423.56,A -85,B 0,C 180,E1 -18555.915,E2 -18555.915} C_VEL
LIN {X 0,Y 256.168,Z 423.573,A -85,B 0,C 180,E1 -18560.895,E2 -18560.895} C_VEL
LIN {X 0,Y 256.19,Z 423.572,A -85,B 0,C 180,E1 -18565.139,E2 -18565.139} C_VEL
LIN {X 0,Y 256.112,Z 423.583,A -85,B 0,C 180,E1 -18569.6,E2 -18569.6} C_VEL
LIN {X 0,Y 256.086,Z 423.585,A -85,B 0,C 180,E1 -18573.29,E2 -18573.29} C_VEL
LIN {X 0,Y 256.13,Z 423.582,A -85,B 0,C 180,E1 -18577.275,E2 -18577.275} C_VEL
LIN {X 0,Y 256.058,Z 423.59,A -85,B 0,C 180,E1 -18581.203,E2 -18581.203} C_VEL
LIN {X 0,Y 256.063,Z 423.59,A -85,B 0,C 180,E1 -18585.529,E2 -18585.529} C_VEL
LIN {X 0,Y 256.058,Z 423.59,A -85,B 0,C 180,E1 -18588.797,E2 -18588.797} C_VEL
LIN {X 0,Y 256.094,Z 423.717,A -85,B 0,C 180,E1 -18590.211,E2 -18590.211} C_VEL
LIN {X 0,Y 256.25,Z 425.699,A -85,B 0,C 180,E1 -18592.888,E2 -18592.888} C_VEL
LIN {X 0,Y 256.112,Z 428.745,A -85,B 0,C 180,E1 -18596.714,E2 -18596.714} C_VEL
LIN {X 0,Y 255.753,Z 431.841,A -85,B 0,C 180,E1 -18600.355,E2 -18600.355} C_VEL
LIN {X 0,Y 255.716,Z 432.498,A -85,B 0,C 180,E1 -18601.104,E2 -18601.104} C_VEL
LIN {X 0,Y 256.701,Z 435.639,A -85,B 0,C 180,E1 -18601.375,E2 -18601.375} C_VEL
LIN {X 0,Y 260.499,Z 446.889,A -85,B 0,C 180,E1 -18602.514,E2 -18602.514} C_VEL
LIN {X 0,Y 263.37,Z 458.099,A -85,B 0,C 180,E1 -18603.786,E2 -18603.786} C_VEL
LIN {X 0,Y 265.58,Z 469.875,A -85,B 0,C 180,E1 -18605.322,E2 -18605.322} C_VEL
LIN {X 0,Y 266.397,Z 476.784,A -85,B 0,C 180,E1 -18606.341,E2 -18606.341} C_VEL
LIN {X 0,Y 264.502,Z 487.902,A -85,B 0,C 180,E1 -18607.957,E2 -18607.957} C_VEL
LIN {X 0,Y 262.829,Z 497.209,A -85,B 0,C 180,E1 -18609.658,E2 -18609.658} C_VEL
LIN {X 0,Y 260.923,Z 505.693,A -85,B 0,C 180,E1 -18611.549,E2 -18611.549} C_VEL
LIN {X 0,Y 258.969,Z 513.94,A -85,B 0,C 180,E1 -18613.849,E2 -18613.849} C_VEL
LIN {X 0,Y 257.372,Z 520.581,A -85,B 0,C 180,E1 -18616.176,E2 -18616.176} C_VEL
LIN {X 0,Y 255.925,Z 526.661,A -85,B 0,C 180,E1 -18618.917,E2 -18618.917} C_VEL
LIN {X 0,Y 255.078,Z 530.607,A -85,B 0,C 180,E1 -18621.284,E2 -18621.284} C_VEL
LIN {X 0,Y 254.514,Z 533.627,A -85,B 0,C 180,E1 -18623.766,E2 -18623.766} C_VEL
LIN {X 0,Y 254.194,Z 535.9,A -85,B 0,C 180,E1 -18626.83,E2 -18626.83} C_VEL
LIN {X 0,Y 254.096,Z 536.509,A -85,B 0,C 180,E1 -18628.415,E2 -18628.415} C_VEL
LIN {X 0,Y 254.063,Z 536.739,A -85,B 0,C 180,E1 -18630,E2 -18630} C_VEL
LIN {X 0,Y 254.095,Z 536.545,A -85,B 0,C 180,E1 -18631.585,E2 -18631.585} C_VEL
LIN {X 0,Y 254.192,Z 535.959,A -85,B 0,C 180,E1 -18633.17,E2 -18633.17} C_VEL
LIN {X 0,Y 254.566,Z 533.636,A -85,B 0,C 180,E1 -18636.34,E2 -18636.34} C_VEL
LIN {X 0,Y 255.077,Z 530.77,A -85,B 0,C 180,E1 -18638.716,E2 -18638.716} C_VEL
LIN {X 0,Y 255.91,Z 526.881,A -85,B 0,C 180,E1 -18641.084,E2 -18641.084} C_VEL
LIN {X 0,Y 257.093,Z 521.861,A -85,B 0,C 180,E1 -18643.436,E2 -18643.436} C_VEL
LIN {X 0,Y 258.543,Z 515.54,A -85,B 0,C 180,E1 -18645.773,E2 -18645.773} C_VEL
LIN {X 0,Y 260.492,Z 507.623,A -85,B 0,C 180,E1 -18648.076,E2 -18648.076} C_VEL
LIN {X 0,Y 262.284,Z 499.554,A -85,B 0,C 180,E1 -18649.977,E2 -18649.977} C_VEL
LIN {X 0,Y 264.181,Z 489.71,A -85,B 0,C 180,E1 -18651.867,E2 -18651.867} C_VEL
LIN {X 0,Y 266.258,Z 478.764,A -85,B 0,C 180,E1 -18653.509,E2 -18653.509} C_VEL
LIN {X 0,Y 266.16,Z 474.946,A -85,B 0,C 180,E1 -18654.075,E2 -18654.075} C_VEL
LIN {X 0,Y 264.759,Z 464.684,A -85,B 0,C 180,E1 -18655.507,E2 -18655.507} C_VEL
LIN {X 0,Y 262.146,Z 452.951,A -85,B 0,C 180,E1 -18656.949,E2 -18656.949} C_VEL
LIN {X 0,Y 258.674,Z 441.069,A -85,B 0,C 180,E1 -18658.219,E2 -18658.219} C_VEL
LIN {X 0,Y 255.829,Z 433.219,A -85,B 0,C 180,E1 -18658.984,E2 -18658.984} C_VEL
LIN {X 0,Y 255.705,Z 432.456,A -85,B 0,C 180,E1 -18659.073,E2 -18659.073} C_VEL
LIN {X 0,Y 256.104,Z 428.86,A -85,B 0,C 180,E1 -18663.288,E2 -18663.288} C_VEL
LIN {X 0,Y 256.239,Z 427.326,A -85,B 0,C 180,E1 -18665.168,E2 -18665.168} C_VEL
LIN {X 0,Y 256.251,Z 425.656,A -85,B 0,C 180,E1 -18667.31,E2 -18667.31} C_VEL
LIN {X 0,Y 256.128,Z 423.811,A -85,B 0,C 180,E1 -18669.798,E2 -18669.798} C_VEL
LIN {X 0,Y 256.067,Z 423.586,A -85,B 0,C 180,E1 -18673.326,E2 -18673.326} C_VEL
LIN {X 0,Y 256.075,Z 423.586,A -85,B 0,C 180,E1 -18677.818,E2 -18677.818} C_VEL
LIN {X 0,Y 256.091,Z 423.585,A -85,B 0,C 180,E1 -18680.861,E2 -18680.861} C_VEL
LIN {X 0,Y 256.123,Z 423.583,A -85,B 0,C 180,E1 -18684.813,E2 -18684.813} C_VEL
LIN {X 0,Y 256.095,Z 423.586,A -85,B 0,C 180,E1 -18688.573,E2 -18688.573} C_VEL
LIN {X 0,Y 256.141,Z 423.58,A -85,B 0,C 180,E1 -18692.196,E2 -18692.196} C_VEL
LIN {X 0,Y 256.171,Z 423.573,A -85,B 0,C 180,E1 -18695.699,E2 -18695.699} C_VEL
LIN {X 0,Y 256.172,Z 423.573,A -85,B 0,C 180,E1 -18699.105,E2 -18699.105} C_VEL
LIN {X 0,Y 256.303,Z 423.561,A -85,B 0,C 180,E1 -18704.085,E2 -18704.085} C_VEL
LIN {X 0,Y 256.313,Z 423.556,A -85,B 0,C 180,E1 -18708.934,E2 -18708.934} C_VEL
LIN {X 0,Y 256.543,Z 423.53,A -85,B 0,C 180,E1 -18712.127,E2 -18712.127} C_VEL
LIN {X 0,Y 256.716,Z 423.506,A -85,B 0,C 180,E1 -18718.431,E2 -18718.431} C_VEL
LIN {X 0,Y 256.717,Z 423.508,A -85,B 0,C 180,E1 -18721.569,E2 -18721.569} C_VEL
LIN {X 0,Y 256.543,Z 423.529,A -85,B 0,C 180,E1 -18727.873,E2 -18727.873} C_VEL
LIN {X 0,Y 256.313,Z 423.556,A -85,B 0,C 180,E1 -18731.066,E2 -18731.066} C_VEL
LIN {X 0,Y 256.303,Z 423.559,A -85,B 0,C 180,E1 -18735.915,E2 -18735.915} C_VEL
LIN {X 0,Y 256.17,Z 423.575,A -85,B 0,C 180,E1 -18740.895,E2 -18740.895} C_VEL
LIN {X 0,Y 256.19,Z 423.574,A -85,B 0,C 180,E1 -18745.138,E2 -18745.138} C_VEL
LIN {X 0,Y 256.104,Z 423.584,A -85,B 0,C 180,E1 -18749.535,E2 -18749.535} C_VEL
LIN {X 0,Y 255.456,Z 423.673,A -85,B 0,C 180,E1 -18750.847,E2 -18750.847} C_VEL
LIN {X 0,Y 252.615,Z 424.03,A -85,B 0,C 180,E1 -18752.986,E2 -18752.986} C_VEL
LIN {X 0,Y 250.18,Z 424.327,A -85,B 0,C 180,E1 -18754.726,E2 -18754.726} C_VEL
LIN {X 0,Y 249.119,Z 424.453,A -85,B 0,C 180,E1 -18756.076,E2 -18756.076} C_VEL
LIN {X 0,Y 249.025,Z 424.463,A -85,B 0,C 180,E1 -18756.534,E2 -18756.534} C_VEL
LIN {X 0,Y 249.034,Z 424.568,A -85,B 0,C 180,E1 -18759.897,E2 -18759.897} C_VEL
LIN {X 0,Y 249.444,Z 427.062,A -85,B 0,C 180,E1 -18762.9,E2 -18762.9} C_VEL
LIN {X 0,Y 250.087,Z 430.665,A -85,B 0,C 180,E1 -18766.942,E2 -18766.942} C_VEL
LIN {X 0,Y 250.553,Z 433.391,A -85,B 0,C 180,E1 -18769.823,E2 -18769.823} C_VEL
LIN {X 0,Y 250.796,Z 436.531,A -85,B 0,C 180,E1 -18772.951,E2 -18772.951} C_VEL
LIN {X 0,Y 250.448,Z 439.628,A -85,B 0,C 180,E1 -18775.858,E2 -18775.858} C_VEL
LIN {X 0,Y 249.532,Z 444.43,A -85,B 0,C 180,E1 -18780.187,E2 -18780.187} C_VEL
LIN {X 0,Y 253.261,Z 458.466,A -85,B 0,C 180,E1 -18781.462,E2 -18781.462} C_VEL
LIN {X 0,Y 255.803,Z 470.843,A -85,B 0,C 180,E1 -18782.805,E2 -18782.805} C_VEL
LIN {X 0,Y 257.306,Z 483.067,A -85,B 0,C 180,E1 -18784.337,E2 -18784.337} C_VEL
LIN {X 0,Y 257.884,Z 493.507,A -85,B 0,C 180,E1 -18785.871,E2 -18785.871} C_VEL
LIN {X 0,Y 257.663,Z 498.681,A -85,B 0,C 180,E1 -18786.703,E2 -18786.703} C_VEL
LIN {X 0,Y 255.281,Z 509.548,A -85,B 0,C 180,E1 -18788.606,E2 -18788.606} C_VEL
LIN {X 0,Y 253.399,Z 518.386,A -85,B 0,C 180,E1 -18790.56,E2 -18790.56} C_VEL
LIN {X 0,Y 251.691,Z 525.683,A -85,B 0,C 180,E1 -18792.532,E2 -18792.532} C_VEL
LIN {X 0,Y 249.96,Z 532.869,A -85,B 0,C 180,E1 -18794.925,E2 -18794.925} C_VEL
LIN {X 0,Y 248.784,Z 537.722,A -85,B 0,C 180,E1 -18796.938,E2 -18796.938} C_VEL
LIN {X 0,Y 247.858,Z 542.444,A -85,B 0,C 180,E1 -18799.379,E2 -18799.379} C_VEL
LIN {X 0,Y 247.268,Z 546.054,A -85,B 0,C 180,E1 -18801.83,E2 -18801.83} C_VEL
LIN {X 0,Y 247.009,Z 547.916,A -85,B 0,C 180,E1 -18803.465,E2 -18803.465} C_VEL
LIN {X 0,Y 246.883,Z 549.314,A -85,B 0,C 180,E1 -18805.101,E2 -18805.101} C_VEL
LIN {X 0,Y 246.865,Z 550.314,A -85,B 0,C 180,E1 -18806.736,E2 -18806.736} C_VEL
LIN {X 0,Y 246.929,Z 550.925,A -85,B 0,C 180,E1 -18808.369,E2 -18808.369} C_VEL
LIN {X 0,Y 246.985,Z 551.139,A -85,B 0,C 180,E1 -18810,E2 -18810} C_VEL
LIN {X 0,Y 246.928,Z 550.916,A -85,B 0,C 180,E1 -18811.631,E2 -18811.631} C_VEL
LIN {X 0,Y 246.864,Z 550.299,A -85,B 0,C 180,E1 -18813.264,E2 -18813.264} C_VEL
LIN {X 0,Y 246.883,Z 549.294,A -85,B 0,C 180,E1 -18814.899,E2 -18814.899} C_VEL
LIN {X 0,Y 247.009,Z 547.887,A -85,B 0,C 180,E1 -18816.535,E2 -18816.535} C_VEL
LIN {X 0,Y 247.425,Z 544.937,A -85,B 0,C 180,E1 -18818.988,E2 -18818.988} C_VEL
LIN {X 0,Y 248.147,Z 540.949,A -85,B 0,C 180,E1 -18821.435,E2 -18821.435} C_VEL
LIN {X 0,Y 249.45,Z 534.821,A -85,B 0,C 180,E1 -18824.272,E2 -18824.272} C_VEL
LIN {X 0,Y 251.128,Z 528.137,A -85,B 0,C 180,E1 -18826.67,E2 -18826.67} C_VEL
LIN {X 0,Y 253.116,Z 519.717,A -85,B 0,C 180,E1 -18829.077,E2 -18829.077} C_VEL
LIN {X 0,Y 254.871,Z 511.336,A -85,B 0,C 180,E1 -18831.006,E2 -18831.006} C_VEL
LIN {X 0,Y 257.176,Z 500.834,A -85,B 0,C 180,E1 -18832.918,E2 -18832.918} C_VEL
LIN {X 0,Y 257.859,Z 497.206,A -85,B 0,C 180,E1 -18833.491,E2 -18833.491} C_VEL
LIN {X 0,Y 257.463,Z 485.707,A -85,B 0,C 180,E1 -18835.259,E2 -18835.259} C_VEL
LIN {X 0,Y 256.385,Z 474.987,A -85,B 0,C 180,E1 -18836.666,E2 -18836.666} C_VEL
LIN {X 0,Y 254.314,Z 463.112,A -85,B 0,C 180,E1 -18838.021,E2 -18838.021} C_VEL
LIN {X 0,Y 251.037,Z 450.086,A -85,B 0,C 180,E1 -18839.294,E2 -18839.294} C_VEL
LIN {X 0,Y 249.54,Z 444.389,A -85,B 0,C 180,E1 -18839.803,E2 -18839.803} C_VEL
LIN {X 0,Y 250.131,Z 441.321,A -85,B 0,C 180,E1 -18842.55,E2 -18842.55} C_VEL
LIN {X 0,Y 250.711,Z 437.976,A -85,B 0,C 180,E1 -18845.616,E2 -18845.616} C_VEL
LIN {X 0,Y 250.74,Z 435.17,A -85,B 0,C 180,E1 -18848.296,E2 -18848.296} C_VEL
LIN {X 0,Y 250.442,Z 432.787,A -85,B 0,C 180,E1 -18850.739,E2 -18850.739} C_VEL
LIN {X 0,Y 249.837,Z 429.13,A -85,B 0,C 180,E1 -18854.689,E2 -18854.689} C_VEL
LIN {X 0,Y 249.113,Z 424.901,A -85,B 0,C 180,E1 -18859.616,E2 -18859.616} C_VEL
LIN {X 0,Y 249.037,Z 424.468,A -85,B 0,C 180,E1 -18860.619,E2 -18860.619} C_VEL
LIN {X 0,Y 249.046,Z 424.468,A -85,B 0,C 180,E1 -18864.922,E2 -18864.922} C_VEL
LIN {X 0,Y 249.048,Z 424.463,A -85,B 0,C 180,E1 -18869.473,E2 -18869.473} C_VEL
LIN {X 0,Y 249.073,Z 424.459,A -85,B 0,C 180,E1 -18873.162,E2 -18873.162} C_VEL
LIN {X 0,Y 249.081,Z 424.46,A -85,B 0,C 180,E1 -18876.733,E2 -18876.733} C_VEL
LIN {X 0,Y 249.112,Z 424.456,A -85,B 0,C 180,E1 -18880.212,E2 -18880.212} C_VEL
LIN {X 0,Y 249.243,Z 424.438,A -85,B 0,C 180,E1 -18883.622,E2 -18883.622} C_VEL
LIN {X 0,Y 249.255,Z 424.438,A -85,B 0,C 180,E1 -18888.617,E2 -18888.617} C_VEL
LIN {X 0,Y 249.486,Z 424.408,A -85,B 0,C 180,E1 -18891.903,E2 -18891.903} C_VEL
LIN {X 0,Y 249.437,Z 424.413,A -85,B 0,C 180,E1 -18896.77,E2 -18896.77} C_VEL
LIN {X 0,Y 249.737,Z 424.377,A -85,B 0,C 180,E1 -18900,E2 -18900} C_VEL
LIN {X 0,Y 249.437,Z 424.412,A -85,B 0,C 180,E1 -18903.23,E2 -18903.23} C_VEL
LIN {X 0,Y 249.486,Z 424.408,A -85,B 0,C 180,E1 -18908.097,E2 -18908.097} C_VEL
LIN {X 0,Y 249.255,Z 424.435,A -85,B 0,C 180,E1 -18911.383,E2 -18911.383} C_VEL
LIN {X 0,Y 249.243,Z 424.438,A -85,B 0,C 180,E1 -18916.378,E2 -18916.378} C_VEL
LIN {X 0,Y 249.088,Z 424.457,A -85,B 0,C 180,E1 -18921.518,E2 -18921.518} C_VEL
LIN {X 0,Y 249.132,Z 424.452,A -85,B 0,C 180,E1 -18925.482,E2 -18925.482} C_VEL
LIN {X 0,Y 249.082,Z 424.457,A -85,B 0,C 180,E1 -18928.992,E2 -18928.992} C_VEL
LIN {X 0,Y 249.037,Z 424.461,A -85,B 0,C 180,E1 -18932.425,E2 -18932.425} C_VEL
LIN {X 0,Y 249.071,Z 424.458,A -85,B 0,C 180,E1 -18936.339,E2 -18936.339} C_VEL
LIN {X 0,Y 249.027,Z 424.464,A -85,B 0,C 180,E1 -18940.474,E2 -18940.474} C_VEL
LIN {X 0,Y 249.009,Z 424.469,A -85,B 0,C 180,E1 -18944.878,E2 -18944.878} C_VEL
LIN {X 0,Y 249.019,Z 424.468,A -85,B 0,C 180,E1 -18947.364,E2 -18947.364} C_VEL
LIN {X 0,Y 249.035,Z 424.495,A -85,B 0,C 180,E1 -18949.638,E2 -18949.638} C_VEL
LIN {X 0,Y 249.188,Z 427.433,A -85,B 0,C 180,E1 -18953.681,E2 -18953.681} C_VEL
LIN {X 0,Y 249.153,Z 428.959,A -85,B 0,C 180,E1 -18955.657,E2 -18955.657} C_VEL
LIN {X 0,Y 248.803,Z 432.058,A -85,B 0,C 180,E1 -18959.439,E2 -18959.439} C_VEL
LIN {X 0,Y 248.744,Z 432.677,A -85,B 0,C 180,E1 -18960.182,E2 -18960.182} C_VEL
LIN {X 0,Y 250.702,Z 438.445,A -85,B 0,C 180,E1 -18960.756,E2 -18960.756} C_VEL
LIN {X 0,Y 254.42,Z 449.67,A -85,B 0,C 180,E1 -18961.992,E2 -18961.992} C_VEL
LIN {X 0,Y 257.24,Z 461.337,A -85,B 0,C 180,E1 -18963.425,E2 -18963.425} C_VEL
LIN {X 0,Y 259.14,Z 472.549,A -85,B 0,C 180,E1 -18964.999,E2 -18964.999} C_VEL
LIN {X 0,Y 259.767,Z 478.288,A -85,B 0,C 180,E1 -18965.892,E2 -18965.892} C_VEL
LIN {X 0,Y 257.737,Z 489.263,A -85,B 0,C 180,E1 -18967.558,E2 -18967.558} C_VEL
LIN {X 0,Y 255.752,Z 499.221,A -85,B 0,C 180,E1 -18969.49,E2 -18969.49} C_VEL
LIN {X 0,Y 253.501,Z 508.857,A -85,B 0,C 180,E1 -18971.827,E2 -18971.827} C_VEL
LIN {X 0,Y 251.51,Z 516.54,A -85,B 0,C 180,E1 -18974.19,E2 -18974.19} C_VEL
LIN {X 0,Y 250.241,Z 521.782,A -85,B 0,C 180,E1 -18976.189,E2 -18976.189} C_VEL
LIN {X 0,Y 248.947,Z 526.867,A -85,B 0,C 180,E1 -18978.603,E2 -18978.603} C_VEL
LIN {X 0,Y 248.067,Z 530.811,A -85,B 0,C 180,E1 -18981.036,E2 -18981.036} C_VEL
LIN {X 0,Y 247.423,Z 534.03,A -85,B 0,C 180,E1 -18983.811,E2 -18983.811} C_VEL
LIN {X 0,Y 247.114,Z 536.104,A -85,B 0,C 180,E1 -18986.739,E2 -18986.739} C_VEL
LIN {X 0,Y 246.993,Z 536.942,A -85,B 0,C 180,E1 -18990,E2 -18990} C_VEL
LIN {X 0,Y 247.006,Z 536.749,A -85,B 0,C 180,E1 -18991.631,E2 -18991.631} C_VEL
LIN {X 0,Y 247.112,Z 536.162,A -85,B 0,C 180,E1 -18993.261,E2 -18993.261} C_VEL
LIN {X 0,Y 247.503,Z 533.839,A -85,B 0,C 180,E1 -18996.522,E2 -18996.522} C_VEL
LIN {X 0,Y 248.067,Z 530.973,A -85,B 0,C 180,E1 -18998.965,E2 -18998.965} C_VEL
LIN {X 0,Y 248.928,Z 527.084,A -85,B 0,C 180,E1 -19001.399,E2 -19001.399} C_VEL
LIN {X 0,Y 250.177,Z 522.064,A -85,B 0,C 180,E1 -19003.815,E2 -19003.815} C_VEL
LIN {X 0,Y 251.725,Z 515.741,A -85,B 0,C 180,E1 -19006.212,E2 -19006.212} C_VEL
LIN {X 0,Y 253.756,Z 507.825,A -85,B 0,C 180,E1 -19008.573,E2 -19008.573} C_VEL
LIN {X 0,Y 255.6,Z 499.805,A -85,B 0,C 180,E1 -19010.511,E2 -19010.511} C_VEL
LIN {X 0,Y 257.618,Z 489.91,A -85,B 0,C 180,E1 -19012.453,E2 -19012.453} C_VEL
LIN {X 0,Y 259.746,Z 479.062,A -85,B 0,C 180,E1 -19014.121,E2 -19014.121} C_VEL
LIN {X 0,Y 258.671,Z 469.24,A -85,B 0,C 180,E1 -19015.619,E2 -19015.619} C_VEL
LIN {X 0,Y 256.575,Z 458.273,A -85,B 0,C 180,E1 -19017.1,E2 -19017.1} C_VEL
LIN {X 0,Y 253.473,Z 446.436,A -85,B 0,C 180,E1 -19018.501,E2 -19018.501} C_VEL
LIN {X 0,Y 249.506,Z 435.393,A -85,B 0,C 180,E1 -19019.691,E2 -19019.691} C_VEL
LIN {X 0,Y 248.739,Z 432.666,A -85,B 0,C 180,E1 -19019.972,E2 -19019.972} C_VEL
LIN {X 0,Y 249.005,Z 430.625,A -85,B 0,C 180,E1 -19022.43,E2 -19022.43} C_VEL
LIN {X 0,Y 249.219,Z 428.447,A -85,B 0,C 180,E1 -19025.134,E2 -19025.134} C_VEL
LIN {X 0,Y 249.174,Z 426.032,A -85,B 0,C 180,E1 -19028.354,E2 -19028.354} C_VEL
LIN {X 0,Y 249.04,Z 424.523,A -85,B 0,C 180,E1 -19030.472,E2 -19030.472} C_VEL
LIN {X 0,Y 249.01,Z 424.467,A -85,B 0,C 180,E1 -19034.878,E2 -19034.878} C_VEL
LIN {X 0,Y 249.02,Z 424.466,A -85,B 0,C 180,E1 -19037.363,E2 -19037.363} C_VEL
LIN {X 0,Y 249.041,Z 424.461,A -85,B 0,C 180,E1 -19041.622,E2 -19041.622} C_VEL
LIN {X 0,Y 249.064,Z 424.46,A -85,B 0,C 180,E1 -19045.642,E2 -19045.642} C_VEL
LIN {X 0,Y 249.05,Z 424.46,A -85,B 0,C 180,E1 -19049.473,E2 -19049.473} C_VEL
LIN {X 0,Y 249.075,Z 424.457,A -85,B 0,C 180,E1 -19053.162,E2 -19053.162} C_VEL
LIN {X 0,Y 249.084,Z 424.457,A -85,B 0,C 180,E1 -19056.733,E2 -19056.733} C_VEL
LIN {X 0,Y 249.115,Z 424.455,A -85,B 0,C 180,E1 -19060.212,E2 -19060.212} C_VEL
LIN {X 0,Y 249.245,Z 424.437,A -85,B 0,C 180,E1 -19063.622,E2 -19063.622} C_VEL
LIN {X 0,Y 249.256,Z 424.436,A -85,B 0,C 180,E1 -19068.617,E2 -19068.617} C_VEL
LIN {X 0,Y 249.487,Z 424.408,A -85,B 0,C 180,E1 -19071.903,E2 -19071.903} C_VEL
LIN {X 0,Y 249.438,Z 424.411,A -85,B 0,C 180,E1 -19076.77,E2 -19076.77} C_VEL
LIN {X 0,Y 249.731,Z 424.378,A -85,B 0,C 180,E1 -19080,E2 -19080} C_VEL
LIN {X 0,Y 249.439,Z 424.412,A -85,B 0,C 180,E1 -19083.23,E2 -19083.23} C_VEL
LIN {X 0,Y 249.487,Z 424.407,A -85,B 0,C 180,E1 -19088.097,E2 -19088.097} C_VEL
LIN {X 0,Y 249.256,Z 424.436,A -85,B 0,C 180,E1 -19091.383,E2 -19091.383} C_VEL
LIN {X 0,Y 249.244,Z 424.437,A -85,B 0,C 180,E1 -19096.378,E2 -19096.378} C_VEL
LIN {X 0,Y 249.09,Z 424.458,A -85,B 0,C 180,E1 -19101.518,E2 -19101.518} C_VEL
LIN {X 0,Y 249.132,Z 424.453,A -85,B 0,C 180,E1 -19105.482,E2 -19105.482} C_VEL
LIN {X 0,Y 249.046,Z 424.458,A -85,B 0,C 180,E1 -19109.523,E2 -19109.523} C_VEL
LIN {X 0,Y 249.032,Z 424.453,A -85,B 0,C 180,E1 -19112.426,E2 -19112.426} C_VEL
LIN {X 0,Y 249.025,Z 424.463,A -85,B 0,C 180,E1 -19116.534,E2 -19116.534} C_VEL
LIN {X 0,Y 248.359,Z 424.714,A -85,B 0,C 180,E1 -19117.883,E2 -19117.883} C_VEL
LIN {X 0,Y 245.645,Z 425.972,A -85,B 0,C 180,E1 -19120.075,E2 -19120.075} C_VEL
LIN {X 0,Y 243.43,Z 427.439,A -85,B 0,C 180,E1 -19121.849,E2 -19121.849} C_VEL
LIN {X 0,Y 242.588,Z 428.639,A -85,B 0,C 180,E1 -19123.215,E2 -19123.215} C_VEL
LIN {X 0,Y 242.576,Z 429.035,A -85,B 0,C 180,E1 -19123.676,E2 -19123.676} C_VEL
LIN {X 0,Y 242.984,Z 431.317,A -85,B 0,C 180,E1 -19126.311,E2 -19126.311} C_VEL
LIN {X 0,Y 243.596,Z 435.255,A -85,B 0,C 180,E1 -19130.6,E2 -19130.6} C_VEL
LIN {X 0,Y 243.705,Z 438.477,A -85,B 0,C 180,E1 -19133.85,E2 -19133.85} C_VEL
LIN {X 0,Y 243.122,Z 441.74,A -85,B 0,C 180,E1 -19136.962,E2 -19136.962} C_VEL
LIN {X 0,Y 242.656,Z 444.188,A -85,B 0,C 180,E1 -19139.239,E2 -19139.239} C_VEL
LIN {X 0,Y 244.419,Z 450.446,A -85,B 0,C 180,E1 -19139.816,E2 -19139.816} C_VEL
LIN {X 0,Y 247.649,Z 463.385,A -85,B 0,C 180,E1 -19141.155,E2 -19141.155} C_VEL
LIN {X 0,Y 249.675,Z 474.711,A -85,B 0,C 180,E1 -19142.51,E2 -19142.51} C_VEL
LIN {X 0,Y 250.88,Z 486.709,A -85,B 0,C 180,E1 -19144.16,E2 -19144.16} C_VEL
LIN {X 0,Y 251.212,Z 497.221,A -85,B 0,C 180,E1 -19145.848,E2 -19145.848} C_VEL
LIN {X 0,Y 249.374,Z 506.353,A -85,B 0,C 180,E1 -19147.419,E2 -19147.419} C_VEL
LIN {X 0,Y 247.449,Z 514.877,A -85,B 0,C 180,E1 -19149.205,E2 -19149.205} C_VEL
LIN {X 0,Y 245.299,Z 524.122,A -85,B 0,C 180,E1 -19151.629,E2 -19151.629} C_VEL
LIN {X 0,Y 243.395,Z 531.551,A -85,B 0,C 180,E1 -19154.079,E2 -19154.079} C_VEL
LIN {X 0,Y 241.83,Z 537.518,A -85,B 0,C 180,E1 -19156.556,E2 -19156.556} C_VEL
LIN {X 0,Y 240.859,Z 542.24,A -85,B 0,C 180,E1 -19159.067,E2 -19159.067} C_VEL
LIN {X 0,Y 240.215,Z 545.85,A -85,B 0,C 180,E1 -19161.588,E2 -19161.588} C_VEL
LIN {X 0,Y 239.952,Z 547.713,A -85,B 0,C 180,E1 -19163.272,E2 -19163.272} C_VEL
LIN {X 0,Y 239.774,Z 549.313,A -85,B 0,C 180,E1 -19165.256,E2 -19165.256} C_VEL
LIN {X 0,Y 239.838,Z 550.721,A -85,B 0,C 180,E1 -19168.321,E2 -19168.321} C_VEL
LIN {X 0,Y 239.893,Z 550.936,A -85,B 0,C 180,E1 -19170,E2 -19170} C_VEL
LIN {X 0,Y 239.838,Z 550.712,A -85,B 0,C 180,E1 -19171.679,E2 -19171.679} C_VEL
LIN {X 0,Y 239.801,Z 549.09,A -85,B 0,C 180,E1 -19175.044,E2 -19175.044} C_VEL
LIN {X 0,Y 239.952,Z 547.682,A -85,B 0,C 180,E1 -19176.728,E2 -19176.728} C_VEL
LIN {X 0,Y 240.39,Z 544.732,A -85,B 0,C 180,E1 -19179.253,E2 -19179.253} C_VEL
LIN {X 0,Y 241.166,Z 540.743,A -85,B 0,C 180,E1 -19181.77,E2 -19181.77} C_VEL
LIN {X 0,Y 242.559,Z 534.615,A -85,B 0,C 180,E1 -19184.686,E2 -19184.686} C_VEL
LIN {X 0,Y 244.283,Z 527.929,A -85,B 0,C 180,E1 -19187.151,E2 -19187.151} C_VEL
LIN {X 0,Y 246.233,Z 520.15,A -85,B 0,C 180,E1 -19189.446,E2 -19189.446} C_VEL
LIN {X 0,Y 248.216,Z 511.128,A -85,B 0,C 180,E1 -19191.597,E2 -19191.597} C_VEL
LIN {X 0,Y 250.631,Z 500.626,A -85,B 0,C 180,E1 -19193.552,E2 -19193.552} C_VEL
LIN {X 0,Y 251.134,Z 496.991,A -85,B 0,C 180,E1 -19194.16,E2 -19194.16} C_VEL
LIN {X 0,Y 250.763,Z 485.266,A -85,B 0,C 180,E1 -19196.014,E2 -19196.014} C_VEL
LIN {X 0,Y 249.504,Z 473.72,A -85,B 0,C 180,E1 -19197.58,E2 -19197.58} C_VEL
LIN {X 0,Y 247.466,Z 462.88,A -85,B 0,C 180,E1 -19198.868,E2 -19198.868} C_VEL
LIN {X 0,Y 244.35,Z 450.262,A -85,B 0,C 180,E1 -19200.156,E2 -19200.156} C_VEL
LIN {X 0,Y 242.654,Z 444.176,A -85,B 0,C 180,E1 -19200.729,E2 -19200.729} C_VEL
LIN {X 0,Y 243.477,Z 440.392,A -85,B 0,C 180,E1 -19204.254,E2 -19204.254} C_VEL
LIN {X 0,Y 243.752,Z 437.281,A -85,B 0,C 180,E1 -19207.264,E2 -19207.264} C_VEL
LIN {X 0,Y 243.598,Z 435.198,A -85,B 0,C 180,E1 -19209.399,E2 -19209.399} C_VEL
LIN {X 0,Y 242.976,Z 431.245,A -85,B 0,C 180,E1 -19213.687,E2 -19213.687} C_VEL
LIN {X 0,Y 242.313,Z 427.451,A -85,B 0,C 180,E1 -19218.157,E2 -19218.157} C_VEL
LIN {X 0,Y 241.985,Z 425.347,A -85,B 0,C 180,E1 -19221.038,E2 -19221.038} C_VEL
LIN {X 0,Y 241.989,Z 425.347,A -85,B 0,C 180,E1 -19224.489,E2 -19224.489} C_VEL
LIN {X 0,Y 241.974,Z 425.346,A -85,B 0,C 180,E1 -19228.48,E2 -19228.48} C_VEL
LIN {X 0,Y 242.003,Z 425.341,A -85,B 0,C 180,E1 -19232.312,E2 -19232.312} C_VEL
LIN {X 0,Y 242.058,Z 425.333,A -85,B 0,C 180,E1 -19236.016,E2 -19236.016} C_VEL
LIN {X 0,Y 242.039,Z 425.335,A -85,B 0,C 180,E1 -19239.608,E2 -19239.608} C_VEL
LIN {X 0,Y 242.164,Z 425.32,A -85,B 0,C 180,E1 -19243.278,E2 -19243.278} C_VEL
LIN {X 0,Y 242.189,Z 425.318,A -85,B 0,C 180,E1 -19248.28,E2 -19248.28} C_VEL
LIN {X 0,Y 242.437,Z 425.285,A -85,B 0,C 180,E1 -19251.666,E2 -19251.666} C_VEL
LIN {X 0,Y 242.261,Z 425.306,A -85,B 0,C 180,E1 -19255.007,E2 -19255.007} C_VEL
LIN {X 0,Y 242.638,Z 425.262,A -85,B 0,C 180,E1 -19258.34,E2 -19258.34} C_VEL
LIN {X 0,Y 242.638,Z 425.26,A -85,B 0,C 180,E1 -19261.66,E2 -19261.66} C_VEL
LIN {X 0,Y 242.43,Z 425.286,A -85,B 0,C 180,E1 -19266.747,E2 -19266.747} C_VEL
LIN {X 0,Y 242.347,Z 425.298,A -85,B 0,C 180,E1 -19270.021,E2 -19270.021} C_VEL
LIN {X 0,Y 242.169,Z 425.318,A -85,B 0,C 180,E1 -19275.141,E2 -19275.141} C_VEL
LIN {X 0,Y 242.075,Z 425.327,A -85,B 0,C 180,E1 -19278.624,E2 -19278.624} C_VEL
LIN {X 0,Y 242.014,Z 425.338,A -85,B 0,C 180,E1 -19282.18,E2 -19282.18} C_VEL
LIN {X 0,Y 242.068,Z 425.333,A -85,B 0,C 180,E1 -19285.838,E2 -19285.838} C_VEL
LIN {X 0,Y 242.03,Z 425.337,A -85,B 0,C 180,E1 -19289.58,E2 -19289.58} C_VEL
LIN {X 0,Y 241.993,Z 425.342,A -85,B 0,C 180,E1 -19293.491,E2 -19293.491} C_VEL
LIN {X 0,Y 242.004,Z 425.341,A -85,B 0,C 180,E1 -19297.58,E2 -19297.58} C_VEL
LIN {X 0,Y 241.945,Z 425.348,A -85,B 0,C 180,E1 -19301.921,E2 -19301.921} C_VEL
LIN {X 0,Y 241.938,Z 425.351,A -85,B 0,C 180,E1 -19306.571,E2 -19306.571} C_VEL
LIN {X 0,Y 241.954,Z 425.348,A -85,B 0,C 180,E1 -19309.045,E2 -19309.045} C_VEL
LIN {X 0,Y 242.176,Z 427.658,A -85,B 0,C 180,E1 -19312.452,E2 -19312.452} C_VEL
LIN {X 0,Y 242.179,Z 429.177,A -85,B 0,C 180,E1 -19314.522,E2 -19314.522} C_VEL
LIN {X 0,Y 241.863,Z 432.28,A -85,B 0,C 180,E1 -19318.464,E2 -19318.464} C_VEL
LIN {X 0,Y 241.804,Z 433.084,A -85,B 0,C 180,E1 -19319.271,E2 -19319.271} C_VEL
LIN {X 0,Y 242.874,Z 436.19,A -85,B 0,C 180,E1 -19319.582,E2 -19319.582} C_VEL
LIN {X 0,Y 247.093,Z 448.15,A -85,B 0,C 180,E1 -19320.946,E2 -19320.946} C_VEL
LIN {X 0,Y 250.209,Z 460.245,A -85,B 0,C 180,E1 -19322.466,E2 -19322.466} C_VEL
LIN {X 0,Y 252.32,Z 472.122,A -85,B 0,C 180,E1 -19324.183,E2 -19324.183} C_VEL
LIN {X 0,Y 253.133,Z 479.601,A -85,B 0,C 180,E1 -19325.389,E2 -19325.389} C_VEL
LIN {X 0,Y 250.967,Z 490.525,A -85,B 0,C 180,E1 -19327.132,E2 -19327.132} C_VEL
LIN {X 0,Y 249.12,Z 499.428,A -85,B 0,C 180,E1 -19328.919,E2 -19328.919} C_VEL
LIN {X 0,Y 246.769,Z 509.064,A -85,B 0,C 180,E1 -19331.313,E2 -19331.313} C_VEL
LIN {X 0,Y 244.68,Z 516.746,A -85,B 0,C 180,E1 -19333.737,E2 -19333.737} C_VEL
LIN {X 0,Y 243.34,Z 521.988,A -85,B 0,C 180,E1 -19335.789,E2 -19335.789} C_VEL
LIN {X 0,Y 241.985,Z 527.072,A -85,B 0,C 180,E1 -19338.27,E2 -19338.27} C_VEL
LIN {X 0,Y 241.039,Z 531.017,A -85,B 0,C 180,E1 -19340.772,E2 -19340.772} C_VEL
LIN {X 0,Y 240.319,Z 534.457,A -85,B 0,C 180,E1 -19343.889,E2 -19343.889} C_VEL
LIN {X 0,Y 240.036,Z 536.308,A -85,B 0,C 180,E1 -19346.643,E2 -19346.643} C_VEL
LIN {X 0,Y 239.924,Z 537.145,A -85,B 0,C 180,E1 -19350,E2 -19350} C_VEL
LIN {X 0,Y 239.919,Z 536.952,A -85,B 0,C 180,E1 -19351.679,E2 -19351.679} C_VEL
LIN {X 0,Y 240.034,Z 536.366,A -85,B 0,C 180,E1 -19353.357,E2 -19353.357} C_VEL
LIN {X 0,Y 240.452,Z 534.043,A -85,B 0,C 180,E1 -19356.714,E2 -19356.714} C_VEL
LIN {X 0,Y 241.038,Z 531.177,A -85,B 0,C 180,E1 -19359.228,E2 -19359.228} C_VEL
LIN {X 0,Y 241.962,Z 527.287,A -85,B 0,C 180,E1 -19361.731,E2 -19361.731} C_VEL
LIN {X 0,Y 243.281,Z 522.267,A -85,B 0,C 180,E1 -19364.215,E2 -19364.215} C_VEL
LIN {X 0,Y 244.923,Z 515.943,A -85,B 0,C 180,E1 -19366.675,E2 -19366.675} C_VEL
LIN {X 0,Y 247.041,Z 508.026,A -85,B 0,C 180,E1 -19369.097,E2 -19369.097} C_VEL
LIN {X 0,Y 249.048,Z 499.542,A -85,B 0,C 180,E1 -19371.189,E2 -19371.189} C_VEL
LIN {X 0,Y 251.078,Z 490.11,A -85,B 0,C 180,E1 -19373.072,E2 -19373.072} C_VEL
LIN {X 0,Y 253.073,Z 479.369,A -85,B 0,C 180,E1 -19374.783,E2 -19374.783} C_VEL
LIN {X 0,Y 251.926,Z 469.37,A -85,B 0,C 180,E1 -19376.366,E2 -19376.366} C_VEL
LIN {X 0,Y 249.747,Z 458.155,A -85,B 0,C 180,E1 -19377.938,E2 -19377.938} C_VEL
LIN {X 0,Y 246.583,Z 446.541,A -85,B 0,C 180,E1 -19379.382,E2 -19379.382} C_VEL
LIN {X 0,Y 242.559,Z 435.588,A -85,B 0,C 180,E1 -19380.632,E2 -19380.632} C_VEL
LIN {X 0,Y 241.79,Z 432.889,A -85,B 0,C 180,E1 -19380.931,E2 -19380.931} C_VEL
LIN {X 0,Y 242.055,Z 430.836,A -85,B 0,C 180,E1 -19383.481,E2 -19383.481} C_VEL
LIN {X 0,Y 242.209,Z 429.146,A -85,B 0,C 180,E1 -19385.663,E2 -19385.663} C_VEL
LIN {X 0,Y 242.167,Z 427.149,A -85,B 0,C 180,E1 -19388.41,E2 -19388.41} C_VEL
LIN {X 0,Y 241.961,Z 425.392,A -85,B 0,C 180,E1 -19390.957,E2 -19390.957} C_VEL
LIN {X 0,Y 241.936,Z 425.346,A -85,B 0,C 180,E1 -19394.201,E2 -19394.201} C_VEL
LIN {X 0,Y 241.946,Z 425.347,A -85,B 0,C 180,E1 -19398.079,E2 -19398.079} C_VEL
LIN {X 0,Y 242.005,Z 425.34,A -85,B 0,C 180,E1 -19402.421,E2 -19402.421} C_VEL
LIN {X 0,Y 241.994,Z 425.34,A -85,B 0,C 180,E1 -19406.509,E2 -19406.509} C_VEL
LIN {X 0,Y 242.016,Z 425.337,A -85,B 0,C 180,E1 -19410.597,E2 -19410.597} C_VEL
LIN {X 0,Y 242.07,Z 425.329,A -85,B 0,C 180,E1 -19414.183,E2 -19414.183} C_VEL
LIN {X 0,Y 242.056,Z 425.335,A -85,B 0,C 180,E1 -19418.297,E2 -19418.297} C_VEL
LIN {X 0,Y 242.166,Z 425.318,A -85,B 0,C 180,E1 -19423.278,E2 -19423.278} C_VEL
LIN {X 0,Y 242.189,Z 425.317,A -85,B 0,C 180,E1 -19428.28,E2 -19428.28} C_VEL
LIN {X 0,Y 242.438,Z 425.284,A -85,B 0,C 180,E1 -19431.666,E2 -19431.666} C_VEL
LIN {X 0,Y 242.262,Z 425.306,A -85,B 0,C 180,E1 -19435.007,E2 -19435.007} C_VEL
LIN {X 0,Y 242.639,Z 425.26,A -85,B 0,C 180,E1 -19438.34,E2 -19438.34} C_VEL
LIN {X 0,Y 242.639,Z 425.263,A -85,B 0,C 180,E1 -19441.66,E2 -19441.66} C_VEL
LIN {X 0,Y 242.437,Z 425.285,A -85,B 0,C 180,E1 -19446.659,E2 -19446.659} C_VEL
LIN {X 0,Y 242.348,Z 425.296,A -85,B 0,C 180,E1 -19450.02,E2 -19450.02} C_VEL
LIN {X 0,Y 242.17,Z 425.32,A -85,B 0,C 180,E1 -19455.141,E2 -19455.141} C_VEL
LIN {X 0,Y 242.076,Z 425.33,A -85,B 0,C 180,E1 -19458.624,E2 -19458.624} C_VEL
LIN {X 0,Y 242.015,Z 425.337,A -85,B 0,C 180,E1 -19462.18,E2 -19462.18} C_VEL
LIN {X 0,Y 242.069,Z 425.331,A -85,B 0,C 180,E1 -19465.838,E2 -19465.838} C_VEL
LIN {X 0,Y 242.009,Z 425.34,A -85,B 0,C 180,E1 -19469.583,E2 -19469.583} C_VEL
LIN {X 0,Y 241.983,Z 425.331,A -85,B 0,C 180,E1 -19473.492,E2 -19473.492} C_VEL
LIN {X 0,Y 241.989,Z 425.342,A -85,B 0,C 180,E1 -19477.582,E2 -19477.582} C_VEL
LIN {X 0,Y 242.027,Z 425.499,A -85,B 0,C 180,E1 -19479.329,E2 -19479.329} C_VEL
LIN {X 0,Y 242.576,Z 429.035,A -85,B 0,C 180,E1 -19483.676,E2 -19483.676} C_VEL
LIN {X 0,Y 242.135,Z 430.315,A -85,B 0,C 180,E1 -19485.033,E2 -19485.033} C_VEL
LIN {X 0,Y 239.671,Z 432.742,A -85,B 0,C 180,E1 -19487.241,E2 -19487.241} C_VEL
LIN {X 0,Y 236.832,Z 435.72,A -85,B 0,C 180,E1 -19489.956,E2 -19489.956} C_VEL
LIN {X 0,Y 236.611,Z 436.635,A -85,B 0,C 180,E1 -19490.894,E2 -19490.894} C_VEL
LIN {X 0,Y 236.691,Z 439.2,A -85,B 0,C 180,E1 -19493.569,E2 -19493.569} C_VEL
LIN {X 0,Y 236.189,Z 442.091,A -85,B 0,C 180,E1 -19496.425,E2 -19496.425} C_VEL
LIN {X 0,Y 235.79,Z 444.147,A -85,B 0,C 180,E1 -19498.273,E2 -19498.273} C_VEL
LIN {X 0,Y 237.744,Z 450.646,A -85,B 0,C 180,E1 -19498.899,E2 -19498.899} C_VEL
LIN {X 0,Y 240.892,Z 463.17,A -85,B 0,C 180,E1 -19500.266,E2 -19500.266} C_VEL
LIN {X 0,Y 242.936,Z 474.499,A -85,B 0,C 180,E1 -19501.68,E2 -19501.68} C_VEL
LIN {X 0,Y 244.098,Z 485.169,A -85,B 0,C 180,E1 -19503.195,E2 -19503.195} C_VEL
LIN {X 0,Y 244.499,Z 495.711,A -85,B 0,C 180,E1 -19504.914,E2 -19504.914} C_VEL
LIN {X 0,Y 244.364,Z 499.455,A -85,B 0,C 180,E1 -19505.579,E2 -19505.579} C_VEL
LIN {X 0,Y 242.075,Z 509.145,A -85,B 0,C 180,E1 -19507.376,E2 -19507.376} C_VEL
LIN {X 0,Y 239.991,Z 517.981,A -85,B 0,C 180,E1 -19509.426,E2 -19509.426} C_VEL
LIN {X 0,Y 238.168,Z 525.278,A -85,B 0,C 180,E1 -19511.505,E2 -19511.505} C_VEL
LIN {X 0,Y 236.235,Z 532.463,A -85,B 0,C 180,E1 -19514.027,E2 -19514.027} C_VEL
LIN {X 0,Y 234.891,Z 537.314,A -85,B 0,C 180,E1 -19516.151,E2 -19516.151} C_VEL
LIN {X 0,Y 233.875,Z 542.037,A -85,B 0,C 180,E1 -19518.736,E2 -19518.736} C_VEL
LIN {X 0,Y 233.182,Z 545.647,A -85,B 0,C 180,E1 -19521.332,E2 -19521.332} C_VEL
LIN {X 0,Y 232.89,Z 547.509,A -85,B 0,C 180,E1 -19523.067,E2 -19523.067} C_VEL
LIN {X 0,Y 232.684,Z 549.278,A -85,B 0,C 180,E1 -19525.368,E2 -19525.368} C_VEL
LIN {X 0,Y 232.749,Z 550.517,A -85,B 0,C 180,E1 -19528.269,E2 -19528.269} C_VEL
LIN {X 0,Y 232.804,Z 550.732,A -85,B 0,C 180,E1 -19530,E2 -19530} C_VEL
LIN {X 0,Y 232.749,Z 550.508,A -85,B 0,C 180,E1 -19531.73,E2 -19531.73} C_VEL
LIN {X 0,Y 232.731,Z 548.885,A -85,B 0,C 180,E1 -19535.198,E2 -19535.198} C_VEL
LIN {X 0,Y 232.89,Z 547.477,A -85,B 0,C 180,E1 -19536.933,E2 -19536.933} C_VEL
LIN {X 0,Y 233.373,Z 544.526,A -85,B 0,C 180,E1 -19539.534,E2 -19539.534} C_VEL
LIN {X 0,Y 234.179,Z 540.537,A -85,B 0,C 180,E1 -19542.127,E2 -19542.127} C_VEL
LIN {X 0,Y 235.676,Z 534.409,A -85,B 0,C 180,E1 -19545.125,E2 -19545.125} C_VEL
LIN {X 0,Y 237.449,Z 527.722,A -85,B 0,C 180,E1 -19547.661,E2 -19547.661} C_VEL
LIN {X 0,Y 239.752,Z 518.994,A -85,B 0,C 180,E1 -19550.275,E2 -19550.275} C_VEL
LIN {X 0,Y 241.609,Z 510.92,A -85,B 0,C 180,E1 -19552.219,E2 -19552.219} C_VEL
LIN {X 0,Y 244.109,Z 500.418,A -85,B 0,C 180,E1 -19554.221,E2 -19554.221} C_VEL
LIN {X 0,Y 244.442,Z 495.473,A -85,B 0,C 180,E1 -19555.092,E2 -19555.092} C_VEL
LIN {X 0,Y 243.972,Z 483.783,A -85,B 0,C 180,E1 -19556.978,E2 -19556.978} C_VEL
LIN {X 0,Y 242.668,Z 472.83,A -85,B 0,C 180,E1 -19558.503,E2 -19558.503} C_VEL
LIN {X 0,Y 240.312,Z 460.661,A -85,B 0,C 180,E1 -19559.977,E2 -19559.977} C_VEL
LIN {X 0,Y 237.173,Z 448.977,A -85,B 0,C 180,E1 -19561.225,E2 -19561.225} C_VEL
LIN {X 0,Y 235.809,Z 443.956,A -85,B 0,C 180,E1 -19561.726,E2 -19561.726} C_VEL
LIN {X 0,Y 236.463,Z 441.201,A -85,B 0,C 180,E1 -19564.382,E2 -19564.382} C_VEL
LIN {X 0,Y 236.704,Z 438.876,A -85,B 0,C 180,E1 -19566.711,E2 -19566.711} C_VEL
LIN {X 0,Y 236.591,Z 436.263,A -85,B 0,C 180,E1 -19569.436,E2 -19569.436} C_VEL
LIN {X 0,Y 236.02,Z 432.858,A -85,B 0,C 180,E1 -19573.226,E2 -19573.226} C_VEL
LIN {X 0,Y 235.34,Z 428.673,A -85,B 0,C 180,E1 -19578.295,E2 -19578.295} C_VEL
LIN {X 0,Y 234.957,Z 426.223,A -85,B 0,C 180,E1 -19581.635,E2 -19581.635} C_VEL
LIN {X 0,Y 234.931,Z 426.225,A -85,B 0,C 180,E1 -19585.362,E2 -19585.362} C_VEL
LIN {X 0,Y 234.923,Z 426.223,A -85,B 0,C 180,E1 -19589.431,E2 -19589.431} C_VEL
LIN {X 0,Y 234.994,Z 426.212,A -85,B 0,C 180,E1 -19593.794,E2 -19593.794} C_VEL
LIN {X 0,Y 235.013,Z 426.213,A -85,B 0,C 180,E1 -19598.97,E2 -19598.97} C_VEL
LIN {X 0,Y 235.098,Z 426.201,A -85,B 0,C 180,E1 -19603.059,E2 -19603.059} C_VEL
LIN {X 0,Y 235.149,Z 426.194,A -85,B 0,C 180,E1 -19607.924,E2 -19607.924} C_VEL
LIN {X 0,Y 235.392,Z 426.162,A -85,B 0,C 180,E1 -19611.415,E2 -19611.415} C_VEL
LIN {X 0,Y 235.407,Z 426.158,A -85,B 0,C 180,E1 -19613.142,E2 -19613.142} C_VEL
LIN {X 0,Y 235.597,Z 426.139,A -85,B 0,C 180,E1 -19618.291,E2 -19618.291} C_VEL
LIN {X 0,Y 235.597,Z 426.138,A -85,B 0,C 180,E1 -19621.71,E2 -19621.71} C_VEL
LIN {X 0,Y 235.407,Z 426.161,A -85,B 0,C 180,E1 -19626.859,E2 -19626.859} C_VEL
LIN {X 0,Y 235.255,Z 426.18,A -85,B 0,C 180,E1 -19630.326,E2 -19630.326} C_VEL
LIN {X 0,Y 235.116,Z 426.199,A -85,B 0,C 180,E1 -19635.606,E2 -19635.606} C_VEL
LIN {X 0,Y 235.01,Z 426.208,A -85,B 0,C 180,E1 -19639.206,E2 -19639.206} C_VEL
LIN {X 0,Y 234.962,Z 426.215,A -85,B 0,C 180,E1 -19642.883,E2 -19642.883} C_VEL
LIN {X 0,Y 234.971,Z 426.214,A -85,B 0,C 180,E1 -19646.657,E2 -19646.657} C_VEL
LIN {X 0,Y 234.933,Z 426.219,A -85,B 0,C 180,E1 -19650.568,E2 -19650.568} C_VEL
LIN {X 0,Y 234.962,Z 426.215,A -85,B 0,C 180,E1 -19654.633,E2 -19654.633} C_VEL
LIN {X 0,Y 234.943,Z 426.22,A -85,B 0,C 180,E1 -19658.945,E2 -19658.945} C_VEL
LIN {X 0,Y 234.891,Z 426.226,A -85,B 0,C 180,E1 -19663.485,E2 -19663.485} C_VEL
LIN {X 0,Y 234.891,Z 426.229,A -85,B 0,C 180,E1 -19666.515,E2 -19666.515} C_VEL
LIN {X 0,Y 234.921,Z 426.369,A -85,B 0,C 180,E1 -19668.84,E2 -19668.84} C_VEL
LIN {X 0,Y 235.087,Z 427.877,A -85,B 0,C 180,E1 -19671.112,E2 -19671.112} C_VEL
LIN {X 0,Y 235.162,Z 429.764,A -85,B 0,C 180,E1 -19673.796,E2 -19673.796} C_VEL
LIN {X 0,Y 234.87,Z 433.12,A -85,B 0,C 180,E1 -19678.232,E2 -19678.232} C_VEL
LIN {X 0,Y 235.957,Z 436.434,A -85,B 0,C 180,E1 -19678.591,E2 -19678.591} C_VEL
LIN {X 0,Y 240.293,Z 448.525,A -85,B 0,C 180,E1 -19680.052,E2 -19680.052} C_VEL
LIN {X 0,Y 243.415,Z 460.342,A -85,B 0,C 180,E1 -19681.615,E2 -19681.615} C_VEL
LIN {X 0,Y 245.285,Z 470.548,A -85,B 0,C 180,E1 -19683.124,E2 -19683.124} C_VEL
LIN {X 0,Y 246.428,Z 479.819,A -85,B 0,C 180,E1 -19684.673,E2 -19684.673} C_VEL
LIN {X 0,Y 245.913,Z 483.725,A -85,B 0,C 180,E1 -19685.294,E2 -19685.294} C_VEL
LIN {X 0,Y 243.952,Z 493.199,A -85,B 0,C 180,E1 -19686.956,E2 -19686.956} C_VEL
LIN {X 0,Y 241.727,Z 503.096,A -85,B 0,C 180,E1 -19689.136,E2 -19689.136} C_VEL
LIN {X 0,Y 239.277,Z 512.004,A -85,B 0,C 180,E1 -19691.594,E2 -19691.594} C_VEL
LIN {X 0,Y 237.305,Z 519.17,A -85,B 0,C 180,E1 -19694.101,E2 -19694.101} C_VEL
LIN {X 0,Y 235.932,Z 524.001,A -85,B 0,C 180,E1 -19696.214,E2 -19696.214} C_VEL
LIN {X 0,Y 234.643,Z 528.694,A -85,B 0,C 180,E1 -19698.774,E2 -19698.774} C_VEL
LIN {X 0,Y 233.794,Z 532.28,A -85,B 0,C 180,E1 -19701.356,E2 -19701.356} C_VEL
LIN {X 0,Y 233.226,Z 534.864,A -85,B 0,C 180,E1 -19703.947,E2 -19703.947} C_VEL
LIN {X 0,Y 232.96,Z 536.512,A -85,B 0,C 180,E1 -19706.541,E2 -19706.541} C_VEL
LIN {X 0,Y 232.835,Z 537.349,A -85,B 0,C 180,E1 -19710,E2 -19710} C_VEL
LIN {X 0,Y 232.835,Z 537.156,A -85,B 0,C 180,E1 -19711.73,E2 -19711.73} C_VEL
LIN {X 0,Y 232.958,Z 536.569,A -85,B 0,C 180,E1 -19713.459,E2 -19713.459} C_VEL
LIN {X 0,Y 233.389,Z 534.246,A -85,B 0,C 180,E1 -19716.918,E2 -19716.918} C_VEL
LIN {X 0,Y 234.031,Z 531.38,A -85,B 0,C 180,E1 -19719.507,E2 -19719.507} C_VEL
LIN {X 0,Y 235.013,Z 527.49,A -85,B 0,C 180,E1 -19722.083,E2 -19722.083} C_VEL
LIN {X 0,Y 236.399,Z 522.469,A -85,B 0,C 180,E1 -19724.638,E2 -19724.638} C_VEL
LIN {X 0,Y 238.13,Z 516.145,A -85,B 0,C 180,E1 -19727.166,E2 -19727.166} C_VEL
LIN {X 0,Y 240.348,Z 508.227,A -85,B 0,C 180,E1 -19729.65,E2 -19729.65} C_VEL
LIN {X 0,Y 242.282,Z 500.364,A -85,B 0,C 180,E1 -19731.655,E2 -19731.655} C_VEL
LIN {X 0,Y 244.554,Z 490.311,A -85,B 0,C 180,E1 -19733.724,E2 -19733.724} C_VEL
LIN {X 0,Y 246.459,Z 480.616,A -85,B 0,C 180,E1 -19735.324,E2 -19735.324} C_VEL
LIN {X 0,Y 245.416,Z 470.958,A -85,B 0,C 180,E1 -19736.936,E2 -19736.936} C_VEL
LIN {X 0,Y 243.342,Z 459.871,A -85,B 0,C 180,E1 -19738.581,E2 -19738.581} C_VEL
LIN {X 0,Y 240.203,Z 448.204,A -85,B 0,C 180,E1 -19740.126,E2 -19740.126} C_VEL
LIN {X 0,Y 235.903,Z 436.353,A -85,B 0,C 180,E1 -19741.564,E2 -19741.564} C_VEL
